LIN {X 0,Y 501.584,Z 1086.03,A -85,B 0,C 180,E1 12402.194,E2 12402.194} C_VEL
LIN {X 0,Y 502.565,Z 1075.07,A -85,B 0,C 180,E1 12406.965,E2 12406.965} C_VEL
LIN {X 0,Y 503.829,Z 1050.291,A -85,B 0,C 180,E1 12410.955,E2 12410.955} C_VEL
LIN {X 0,Y 505.175,Z 1014.827,A -85,B 0,C 180,E1 12413.746,E2 12413.746} C_VEL
LIN {X 0,Y 505.31,Z 972.689,A -85,B 0,C 180,E1 12415.098,E2 12415.098} C_VEL
LIN {X 0,Y 507.178,Z 860.099,A -85,B 0,C 180,E1 12417.103,E2 12417.103} C_VEL
LIN {X 0,Y 506.379,Z 795.398,A -85,B 0,C 180,E1 12419.992,E2 12419.992} C_VEL
LIN {X 0,Y 498.666,Z 762.06,A -85,B 0,C 180,E1 12422.013,E2 12422.013} C_VEL
LIN {X 0,Y 498.356,Z 762.06,A -85,B 0,C 180,E1 12431.466,E2 12431.466} C_VEL
LIN {X 0,Y 497.906,Z 762.06,A -85,B 0,C 180,E1 12441.773,E2 12441.773} C_VEL
LIN {X 0,Y 497.963,Z 763.805,A -85,B 0,C 180,E1 12445.471,E2 12445.471} C_VEL
LIN {X 0,Y 531.796,Z 813.89,A -85,B 0,C 180,E1 12453.677,E2 12453.677} C_VEL
LIN {X 0,Y 563.025,Z 870.759,A -85,B 0,C 180,E1 12459.883,E2 12459.883} C_VEL
LIN {X 0,Y 551.168,Z 956.836,A -85,B 0,C 180,E1 12463.133,E2 12463.133} C_VEL
LIN {X 0,Y 538.131,Z 1030.007,A -85,B 0,C 180,E1 12467.654,E2 12467.654} C_VEL
LIN {X 0,Y 525.784,Z 1080.484,A -85,B 0,C 180,E1 12472.6,E2 12472.6} C_VEL
LIN {X 0,Y 511.244,Z 1133.404,A -85,B 0,C 180,E1 12480.517,E2 12480.517} C_VEL
LIN {X 0,Y 502.991,Z 1174.818,A -85,B 0,C 180,E1 12489.75,E2 12489.75} C_VEL
LIN {X 0,Y 501.524,Z 1182.015,A -85,B 0,C 180,E1 12491.879,E2 12491.879} C_VEL
LIN {X 0,Y 492.392,Z 1193.006,A -85,B 0,C 180,E1 12495.627,E2 12495.627} C_VEL
LIN {X 0,Y 491.324,Z 1206.842,A -85,B 0,C 180,E1 12503.842,E2 12503.842} C_VEL
LIN {X 0,Y 491.082,Z 1209.864,A -85,B 0,C 180,E1 12510.932,E2 12510.932} C_VEL
LIN {X 0,Y 491.288,Z 1203.601,A -85,B 0,C 180,E1 12518.82,E2 12518.82} C_VEL
LIN {X 0,Y 493.711,Z 1183.881,A -85,B 0,C 180,E1 12527.78,E2 12527.78} C_VEL
LIN {X 0,Y 500.688,Z 1147.15,A -85,B 0,C 180,E1 12537.333,E2 12537.333} C_VEL
LIN {X 0,Y 514.987,Z 1096.477,A -85,B 0,C 180,E1 12546.035,E2 12546.035} C_VEL
LIN {X 0,Y 527.863,Z 1049.194,A -85,B 0,C 180,E1 12551.332,E2 12551.332} C_VEL
LIN {X 0,Y 540.974,Z 981.301,A -85,B 0,C 180,E1 12556.165,E2 12556.165} C_VEL
LIN {X 0,Y 554.262,Z 895.088,A -85,B 0,C 180,E1 12559.986,E2 12559.986} C_VEL
LIN {X 0,Y 555.637,Z 872.387,A -85,B 0,C 180,E1 12560.872,E2 12560.872} C_VEL
LIN {X 0,Y 528.213,Z 820.162,A -85,B 0,C 180,E1 12566.62,E2 12566.62} C_VEL
LIN {X 0,Y 497.316,Z 774.259,A -85,B 0,C 180,E1 12574.21,E2 12574.21} C_VEL
LIN {X 0,Y 489.979,Z 762.06,A -85,B 0,C 180,E1 12576.679,E2 12576.679} C_VEL
LIN {X 0,Y 490.167,Z 762.06,A -85,B 0,C 180,E1 12586.523,E2 12586.523} C_VEL
LIN {X 0,Y 490.448,Z 762.06,A -85,B 0,C 180,E1 12595.512,E2 12595.512} C_VEL
LIN {X 0,Y 490.543,Z 762.06,A -85,B 0,C 180,E1 12602.607,E2 12602.607} C_VEL
LIN {X 0,Y 490.241,Z 762.06,A -85,B 0,C 180,E1 12611.552,E2 12611.552} C_VEL
LIN {X 0,Y 489.948,Z 762.06,A -85,B 0,C 180,E1 12620.807,E2 12620.807} C_VEL
LIN {X 0,Y 490.069,Z 763.934,A -85,B 0,C 180,E1 12627.224,E2 12627.224} C_VEL
LIN {X 0,Y 516.661,Z 805.185,A -85,B 0,C 180,E1 12634.3,E2 12634.3} C_VEL
LIN {X 0,Y 534.44,Z 841.356,A -85,B 0,C 180,E1 12638.266,E2 12638.266} C_VEL
LIN {X 0,Y 545.43,Z 875.323,A -85,B 0,C 180,E1 12641.217,E2 12641.217} C_VEL
LIN {X 0,Y 533.055,Z 952.563,A -85,B 0,C 180,E1 12645.091,E2 12645.091} C_VEL
LIN {X 0,Y 517.932,Z 1030.736,A -85,B 0,C 180,E1 12651.287,E2 12651.287} C_VEL
LIN {X 0,Y 507.374,Z 1083.929,A -85,B 0,C 180,E1 12657.378,E2 12657.378} C_VEL
LIN {X 0,Y 498.428,Z 1126.212,A -85,B 0,C 180,E1 12664.723,E2 12664.723} C_VEL
LIN {X 0,Y 493.224,Z 1157.477,A -85,B 0,C 180,E1 12673.418,E2 12673.418} C_VEL
LIN {X 0,Y 491.274,Z 1174.671,A -85,B 0,C 180,E1 12681.963,E2 12681.963} C_VEL
LIN {X 0,Y 490.815,Z 1179.89,A -85,B 0,C 180,E1 12689.067,E2 12689.067} C_VEL
LIN {X 0,Y 491.301,Z 1175.791,A -85,B 0,C 180,E1 12697.049,E2 12697.049} C_VEL
LIN {X 0,Y 492.893,Z 1158.688,A -85,B 0,C 180,E1 12706.036,E2 12706.036} C_VEL
LIN {X 0,Y 497.85,Z 1128.291,A -85,B 0,C 180,E1 12714.725,E2 12714.725} C_VEL
LIN {X 0,Y 506.517,Z 1087.158,A -85,B 0,C 180,E1 12722.068,E2 12722.068} C_VEL
LIN {X 0,Y 517.427,Z 1033.436,A -85,B 0,C 180,E1 12728.362,E2 12728.362} C_VEL
LIN {X 0,Y 532.611,Z 955.706,A -85,B 0,C 180,E1 12734.592,E2 12734.592} C_VEL
LIN {X 0,Y 544.85,Z 880.188,A -85,B 0,C 180,E1 12738.499,E2 12738.499} C_VEL
LIN {X 0,Y 544.549,Z 868.405,A -85,B 0,C 180,E1 12739.16,E2 12739.16} C_VEL
LIN {X 0,Y 532.956,Z 841.944,A -85,B 0,C 180,E1 12741.803,E2 12741.803} C_VEL
LIN {X 0,Y 506.021,Z 868.419,A -85,B 0,C 180,E1 12744.215,E2 12744.215} C_VEL
LIN {X 0,Y 501.208,Z 875.563,A -85,B 0,C 180,E1 12744.507,E2 12744.507} C_VEL
LIN {X 0,Y 498.271,Z 876.326,A -85,B 0,C 180,E1 12745.014,E2 12745.014} C_VEL
LIN {X 0,Y 497.611,Z 997.367,A -85,B 0,C 180,E1 12747.209,E2 12747.209} C_VEL
LIN {X 0,Y 496.416,Z 1036.646,A -85,B 0,C 180,E1 12749.609,E2 12749.609} C_VEL
LIN {X 0,Y 494.731,Z 1066.862,A -85,B 0,C 180,E1 12753.356,E2 12753.356} C_VEL
LIN {X 0,Y 493.625,Z 1084.009,A -85,B 0,C 180,E1 12757.937,E2 12757.937} C_VEL
LIN {X 0,Y 493.732,Z 1086.304,A -85,B 0,C 180,E1 12763.08,E2 12763.08} C_VEL
LIN {X 0,Y 494.952,Z 1073.478,A -85,B 0,C 180,E1 12767.662,E2 12767.662} C_VEL
LIN {X 0,Y 496.219,Z 1046.852,A -85,B 0,C 180,E1 12771.59,E2 12771.59} C_VEL
LIN {X 0,Y 497.463,Z 1009.558,A -85,B 0,C 180,E1 12774.253,E2 12774.253} C_VEL
LIN {X 0,Y 497.511,Z 956.973,A -85,B 0,C 180,E1 12775.569,E2 12775.569} C_VEL
LIN {X 0,Y 499.597,Z 860.338,A -85,B 0,C 180,E1 12777.386,E2 12777.386} C_VEL
LIN {X 0,Y 498.988,Z 797.899,A -85,B 0,C 180,E1 12780.197,E2 12780.197} C_VEL
LIN {X 0,Y 490.711,Z 762.06,A -85,B 0,C 180,E1 12782.321,E2 12782.321} C_VEL
LIN {X 0,Y 490.334,Z 762.06,A -85,B 0,C 180,E1 12791.656,E2 12791.656} C_VEL
LIN {X 0,Y 489.914,Z 762.06,A -85,B 0,C 180,E1 12800.92,E2 12800.92} C_VEL
LIN {X 0,Y 489.97,Z 764.004,A -85,B 0,C 180,E1 12803.605,E2 12803.605} C_VEL
LIN {X 0,Y 519.882,Z 807.672,A -85,B 0,C 180,E1 12811.563,E2 12811.563} C_VEL
LIN {X 0,Y 553.961,Z 866.925,A -85,B 0,C 180,E1 12818.709,E2 12818.709} C_VEL
LIN {X 0,Y 556.724,Z 877.922,A -85,B 0,C 180,E1 12819.496,E2 12819.496} C_VEL
LIN {X 0,Y 544.196,Z 963.495,A -85,B 0,C 180,E1 12822.887,E2 12822.887} C_VEL
LIN {X 0,Y 530.49,Z 1037.128,A -85,B 0,C 180,E1 12827.636,E2 12827.636} C_VEL
LIN {X 0,Y 517.97,Z 1086.972,A -85,B 0,C 180,E1 12832.705,E2 12832.705} C_VEL
LIN {X 0,Y 502.88,Z 1138.745,A -85,B 0,C 180,E1 12840.976,E2 12840.976} C_VEL
LIN {X 0,Y 494.619,Z 1177.946,A -85,B 0,C 180,E1 12850.328,E2 12850.328} C_VEL
LIN {X 0,Y 492.392,Z 1193.006,A -85,B 0,C 180,E1 12855.627,E2 12855.627} C_VEL
LIN {X 0,Y 483.384,Z 1201.302,A -85,B 0,C 180,E1 12859.554,E2 12859.554} C_VEL
LIN {X 0,Y 483.111,Z 1209.384,A -85,B 0,C 180,E1 12867.348,E2 12867.348} C_VEL
LIN {X 0,Y 483.181,Z 1208.302,A -85,B 0,C 180,E1 12874.551,E2 12874.551} C_VEL
LIN {X 0,Y 483.898,Z 1196.27,A -85,B 0,C 180,E1 12883.159,E2 12883.159} C_VEL
LIN {X 0,Y 487.499,Z 1171.343,A -85,B 0,C 180,E1 12891.983,E2 12891.983} C_VEL
LIN {X 0,Y 498.347,Z 1129.563,A -85,B 0,C 180,E1 12901.42,E2 12901.42} C_VEL
LIN {X 0,Y 512.486,Z 1084.261,A -85,B 0,C 180,E1 12908.318,E2 12908.318} C_VEL
LIN {X 0,Y 526.188,Z 1028.475,A -85,B 0,C 180,E1 12913.62,E2 12913.62} C_VEL
LIN {X 0,Y 540.049,Z 953.551,A -85,B 0,C 180,E1 12918.185,E2 12918.185} C_VEL
LIN {X 0,Y 549.932,Z 876.36,A -85,B 0,C 180,E1 12921.343,E2 12921.343} C_VEL
LIN {X 0,Y 523.592,Z 825.389,A -85,B 0,C 180,E1 12927.097,E2 12927.097} C_VEL
LIN {X 0,Y 491.459,Z 776.33,A -85,B 0,C 180,E1 12935.431,E2 12935.431} C_VEL
LIN {X 0,Y 481.93,Z 762.06,A -85,B 0,C 180,E1 12938.717,E2 12938.717} C_VEL
LIN {X 0,Y 482.263,Z 762.06,A -85,B 0,C 180,E1 12948.146,E2 12948.146} C_VEL
LIN {X 0,Y 483.376,Z 762.06,A -85,B 0,C 180,E1 12959.048,E2 12959.048} C_VEL
LIN {X 0,Y 482.371,Z 762.06,A -85,B 0,C 180,E1 12969.908,E2 12969.908} C_VEL
LIN {X 0,Y 481.917,Z 762.06,A -85,B 0,C 180,E1 12979.248,E2 12979.248} C_VEL
LIN {X 0,Y 482.085,Z 763.893,A -85,B 0,C 180,E1 12985.251,E2 12985.251} C_VEL
LIN {X 0,Y 507.292,Z 802.31,A -85,B 0,C 180,E1 12992.639,E2 12992.639} C_VEL
LIN {X 0,Y 528.284,Z 842.326,A -85,B 0,C 180,E1 12997.503,E2 12997.503} C_VEL
LIN {X 0,Y 539.646,Z 877.144,A -85,B 0,C 180,E1 13000.663,E2 13000.663} C_VEL
LIN {X 0,Y 526.655,Z 954.407,A -85,B 0,C 180,E1 13004.611,E2 13004.611} C_VEL
LIN {X 0,Y 511.633,Z 1026.558,A -85,B 0,C 180,E1 13010.465,E2 13010.465} C_VEL
LIN {X 0,Y 499.546,Z 1085.365,A -85,B 0,C 180,E1 13017.24,E2 13017.24} C_VEL
LIN {X 0,Y 490.459,Z 1127.891,A -85,B 0,C 180,E1 13024.773,E2 13024.773} C_VEL
LIN {X 0,Y 485.168,Z 1158.664,A -85,B 0,C 180,E1 13033.602,E2 13033.602} C_VEL
LIN {X 0,Y 483.157,Z 1175.781,A -85,B 0,C 180,E1 13042.735,E2 13042.735} C_VEL
LIN {X 0,Y 483.141,Z 1179.887,A -85,B 0,C 180,E1 13050.852,E2 13050.852} C_VEL
LIN {X 0,Y 483.496,Z 1173.458,A -85,B 0,C 180,E1 13059.041,E2 13059.041} C_VEL
LIN {X 0,Y 485.186,Z 1154.94,A -85,B 0,C 180,E1 13067.662,E2 13067.662} C_VEL
LIN {X 0,Y 490.529,Z 1125.881,A -85,B 0,C 180,E1 13075.61,E2 13075.61} C_VEL
LIN {X 0,Y 499.831,Z 1082.617,A -85,B 0,C 180,E1 13083.082,E2 13083.082} C_VEL
LIN {X 0,Y 513.288,Z 1018.663,A -85,B 0,C 180,E1 13090.211,E2 13090.211} C_VEL
LIN {X 0,Y 527.819,Z 949.258,A -85,B 0,C 180,E1 13095.598,E2 13095.598} C_VEL
LIN {X 0,Y 539.307,Z 873.653,A -85,B 0,C 180,E1 13099.476,E2 13099.476} C_VEL
LIN {X 0,Y 529.886,Z 852.055,A -85,B 0,C 180,E1 13101.738,E2 13101.738} C_VEL
LIN {X 0,Y 506.285,Z 877.046,A -85,B 0,C 180,E1 13103.639,E2 13103.639} C_VEL
LIN {X 0,Y 497.175,Z 888.251,A -85,B 0,C 180,E1 13104.285,E2 13104.285} C_VEL
LIN {X 0,Y 492.723,Z 893.46,A -85,B 0,C 180,E1 13104.612,E2 13104.612} C_VEL
LIN {X 0,Y 490.436,Z 893.427,A -85,B 0,C 180,E1 13105.053,E2 13105.053} C_VEL
LIN {X 0,Y 489.824,Z 998.567,A -85,B 0,C 180,E1 13107.027,E2 13107.027} C_VEL
LIN {X 0,Y 488.596,Z 1038.169,A -85,B 0,C 180,E1 13109.498,E2 13109.498} C_VEL
LIN {X 0,Y 486.867,Z 1067.564,A -85,B 0,C 180,E1 13113.195,E2 13113.195} C_VEL
LIN {X 0,Y 485.76,Z 1084.332,A -85,B 0,C 180,E1 13117.561,E2 13117.561} C_VEL
LIN {X 0,Y 485.758,Z 1088.321,A -85,B 0,C 180,E1 13122.154,E2 13122.154} C_VEL
LIN {X 0,Y 486.785,Z 1077.934,A -85,B 0,C 180,E1 13126.994,E2 13126.994} C_VEL
LIN {X 0,Y 488.158,Z 1053.73,A -85,B 0,C 180,E1 13131.113,E2 13131.113} C_VEL
LIN {X 0,Y 489.686,Z 1018.309,A -85,B 0,C 180,E1 13134.05,E2 13134.05} C_VEL
LIN {X 0,Y 489.837,Z 975.895,A -85,B 0,C 180,E1 13135.5,E2 13135.5} C_VEL
LIN {X 0,Y 491.945,Z 862.053,A -85,B 0,C 180,E1 13137.621,E2 13137.621} C_VEL
LIN {X 0,Y 491.271,Z 799.056,A -85,B 0,C 180,E1 13140.485,E2 13140.485} C_VEL
LIN {X 0,Y 482.773,Z 762.06,A -85,B 0,C 180,E1 13142.755,E2 13142.755} C_VEL
LIN {X 0,Y 482.347,Z 762.06,A -85,B 0,C 180,E1 13151.852,E2 13151.852} C_VEL
LIN {X 0,Y 482.079,Z 764.083,A -85,B 0,C 180,E1 13161.564,E2 13161.564} C_VEL
LIN {X 0,Y 509.701,Z 804.062,A -85,B 0,C 180,E1 13169.658,E2 13169.658} C_VEL
LIN {X 0,Y 541.657,Z 858.159,A -85,B 0,C 180,E1 13176.848,E2 13176.848} C_VEL
LIN {X 0,Y 551.008,Z 880.185,A -85,B 0,C 180,E1 13178.953,E2 13178.953} C_VEL
LIN {X 0,Y 538.11,Z 964.302,A -85,B 0,C 180,E1 13182.341,E2 13182.341} C_VEL
LIN {X 0,Y 523.928,Z 1038.662,A -85,B 0,C 180,E1 13187.171,E2 13187.171} C_VEL
LIN {X 0,Y 510.351,Z 1092.222,A -85,B 0,C 180,E1 13192.688,E2 13192.688} C_VEL
LIN {X 0,Y 495.736,Z 1139.267,A -85,B 0,C 180,E1 13200.463,E2 13200.463} C_VEL
LIN {X 0,Y 486.53,Z 1179.412,A -85,B 0,C 180,E1 13210.462,E2 13210.462} C_VEL
LIN {X 0,Y 483.384,Z 1201.302,A -85,B 0,C 180,E1 13219.554,E2 13219.554} C_VEL
LIN {X 0,Y 475.339,Z 1206.85,A -85,B 0,C 180,E1 13223.646,E2 13223.646} C_VEL
LIN {X 0,Y 475.092,Z 1209.864,A -85,B 0,C 180,E1 13230.964,E2 13230.964} C_VEL
LIN {X 0,Y 475.378,Z 1203.447,A -85,B 0,C 180,E1 13239.232,E2 13239.232} C_VEL
LIN {X 0,Y 478.01,Z 1183.458,A -85,B 0,C 180,E1 13248.558,E2 13248.558} C_VEL
LIN {X 0,Y 486.538,Z 1146.276,A -85,B 0,C 180,E1 13258.706,E2 13258.706} C_VEL
LIN {X 0,Y 500.843,Z 1102.147,A -85,B 0,C 180,E1 13266.625,E2 13266.625} C_VEL
LIN {X 0,Y 515.281,Z 1049.016,A -85,B 0,C 180,E1 13272.527,E2 13272.527} C_VEL
LIN {X 0,Y 529.378,Z 979.214,A -85,B 0,C 180,E1 13277.472,E2 13277.472} C_VEL
LIN {X 0,Y 543.809,Z 890.869,A -85,B 0,C 180,E1 13281.365,E2 13281.365} C_VEL
LIN {X 0,Y 543.58,Z 878.558,A -85,B 0,C 180,E1 13281.993,E2 13281.993} C_VEL
LIN {X 0,Y 517.866,Z 828.802,A -85,B 0,C 180,E1 13287.841,E2 13287.841} C_VEL
LIN {X 0,Y 488.085,Z 783.083,A -85,B 0,C 180,E1 13295.863,E2 13295.863} C_VEL
LIN {X 0,Y 474.006,Z 762.06,A -85,B 0,C 180,E1 13301.263,E2 13301.263} C_VEL
LIN {X 0,Y 474.607,Z 762.06,A -85,B 0,C 180,E1 13311.675,E2 13311.675} C_VEL
LIN {X 0,Y 474.788,Z 762.06,A -85,B 0,C 180,E1 13320.862,E2 13320.862} C_VEL
LIN {X 0,Y 474.336,Z 762.06,A -85,B 0,C 180,E1 13330.078,E2 13330.078} C_VEL
LIN {X 0,Y 473.886,Z 762.06,A -85,B 0,C 180,E1 13339.587,E2 13339.587} C_VEL
LIN {X 0,Y 474.239,Z 764.161,A -85,B 0,C 180,E1 13343.078,E2 13343.078} C_VEL
LIN {X 0,Y 496.893,Z 797.841,A -85,B 0,C 180,E1 13350.511,E2 13350.511} C_VEL
LIN {X 0,Y 521.962,Z 842.457,A -85,B 0,C 180,E1 13356.636,E2 13356.636} C_VEL
LIN {X 0,Y 533.487,Z 882.016,A -85,B 0,C 180,E1 13360.213,E2 13360.213} C_VEL
LIN {X 0,Y 520.1,Z 957.236,A -85,B 0,C 180,E1 13364.177,E2 13364.177} C_VEL
LIN {X 0,Y 504.516,Z 1028.314,A -85,B 0,C 180,E1 13370.104,E2 13370.104} C_VEL
LIN {X 0,Y 490.514,Z 1092.461,A -85,B 0,C 180,E1 13377.966,E2 13377.966} C_VEL
LIN {X 0,Y 481.795,Z 1133.783,A -85,B 0,C 180,E1 13385.831,E2 13385.831} C_VEL
LIN {X 0,Y 476.551,Z 1162.076,A -85,B 0,C 180,E1 13394.721,E2 13394.721} C_VEL
LIN {X 0,Y 475.121,Z 1176.829,A -85,B 0,C 180,E1 13403.533,E2 13403.533} C_VEL
LIN {X 0,Y 475.143,Z 1179.884,A -85,B 0,C 180,E1 13410.866,E2 13410.866} C_VEL
LIN {X 0,Y 475.482,Z 1173.46,A -85,B 0,C 180,E1 13419.195,E2 13419.195} C_VEL
LIN {X 0,Y 477.332,Z 1154.919,A -85,B 0,C 180,E1 13427.962,E2 13427.962} C_VEL
LIN {X 0,Y 482.786,Z 1126.013,A -85,B 0,C 180,E1 13435.891,E2 13435.891} C_VEL
LIN {X 0,Y 491.966,Z 1083.974,A -85,B 0,C 180,E1 13443.208,E2 13443.208} C_VEL
LIN {X 0,Y 507.71,Z 1014.23,A -85,B 0,C 180,E1 13451.19,E2 13451.19} C_VEL
LIN {X 0,Y 523.097,Z 943.562,A -85,B 0,C 180,E1 13456.57,E2 13456.57} C_VEL
LIN {X 0,Y 533.311,Z 877.091,A -85,B 0,C 180,E1 13459.996,E2 13459.996} C_VEL
LIN {X 0,Y 528.067,Z 863.615,A -85,B 0,C 180,E1 13461.385,E2 13461.385} C_VEL
LIN {X 0,Y 510.923,Z 878.726,A -85,B 0,C 180,E1 13462.864,E2 13462.864} C_VEL
LIN {X 0,Y 484.538,Z 909.606,A -85,B 0,C 180,E1 13464.663,E2 13464.663} C_VEL
LIN {X 0,Y 482.579,Z 910.345,A -85,B 0,C 180,E1 13465.086,E2 13465.086} C_VEL
LIN {X 0,Y 481.993,Z 1000.898,A -85,B 0,C 180,E1 13466.888,E2 13466.888} C_VEL
LIN {X 0,Y 480.759,Z 1040.245,A -85,B 0,C 180,E1 13469.439,E2 13469.439} C_VEL
LIN {X 0,Y 478.974,Z 1069.26,A -85,B 0,C 180,E1 13473.203,E2 13473.203} C_VEL
LIN {X 0,Y 477.843,Z 1085.779,A -85,B 0,C 180,E1 13477.686,E2 13477.686} C_VEL
LIN {X 0,Y 477.87,Z 1089.18,A -85,B 0,C 180,E1 13482.501,E2 13482.501} C_VEL
LIN {X 0,Y 479.093,Z 1077.535,A -85,B 0,C 180,E1 13487.479,E2 13487.479} C_VEL
LIN {X 0,Y 480.432,Z 1053.615,A -85,B 0,C 180,E1 13491.426,E2 13491.426} C_VEL
LIN {X 0,Y 481.967,Z 1016.81,A -85,B 0,C 180,E1 13494.407,E2 13494.407} C_VEL
LIN {X 0,Y 482.09,Z 971.149,A -85,B 0,C 180,E1 13495.823,E2 13495.823} C_VEL
LIN {X 0,Y 484.377,Z 862.498,A -85,B 0,C 180,E1 13497.921,E2 13497.921} C_VEL
LIN {X 0,Y 483.697,Z 800.495,A -85,B 0,C 180,E1 13500.769,E2 13500.769} C_VEL
LIN {X 0,Y 474.792,Z 762.06,A -85,B 0,C 180,E1 13503.03,E2 13503.03} C_VEL
LIN {X 0,Y 474.221,Z 762.06,A -85,B 0,C 180,E1 13513.94,E2 13513.94} C_VEL
LIN {X 0,Y 474.16,Z 764.052,A -85,B 0,C 180,E1 13519.268,E2 13519.268} C_VEL
LIN {X 0,Y 499.405,Z 800.487,A -85,B 0,C 180,E1 13527.536,E2 13527.536} C_VEL
LIN {X 0,Y 530.576,Z 851.548,A -85,B 0,C 180,E1 13535.094,E2 13535.094} C_VEL
LIN {X 0,Y 545.17,Z 883.431,A -85,B 0,C 180,E1 13538.433,E2 13538.433} C_VEL
LIN {X 0,Y 531.635,Z 967.954,A -85,B 0,C 180,E1 13541.934,E2 13541.934} C_VEL
LIN {X 0,Y 517.137,Z 1040.86,A -85,B 0,C 180,E1 13546.77,E2 13546.77} C_VEL
LIN {X 0,Y 503.154,Z 1094.857,A -85,B 0,C 180,E1 13552.402,E2 13552.402} C_VEL
LIN {X 0,Y 489.557,Z 1136.821,A -85,B 0,C 180,E1 13559.298,E2 13559.298} C_VEL
LIN {X 0,Y 479.255,Z 1177.597,A -85,B 0,C 180,E1 13569.511,E2 13569.511} C_VEL
LIN {X 0,Y 475.526,Z 1200.714,A -85,B 0,C 180,E1 13579.012,E2 13579.012} C_VEL
LIN {X 0,Y 475.339,Z 1206.85,A -85,B 0,C 180,E1 13583.646,E2 13583.646} C_VEL
LIN {X 0,Y 467.171,Z 1209.532,A -85,B 0,C 180,E1 13587.823,E2 13587.823} C_VEL
LIN {X 0,Y 467.187,Z 1206.739,A -85,B 0,C 180,E1 13596.577,E2 13596.577} C_VEL
LIN {X 0,Y 468.325,Z 1193.121,A -85,B 0,C 180,E1 13605.073,E2 13605.073} C_VEL
LIN {X 0,Y 474.782,Z 1163.434,A -85,B 0,C 180,E1 13615.109,E2 13615.109} C_VEL
LIN {X 0,Y 488.029,Z 1122.377,A -85,B 0,C 180,E1 13624.124,E2 13624.124} C_VEL
LIN {X 0,Y 502.523,Z 1073.709,A -85,B 0,C 180,E1 13630.693,E2 13630.693} C_VEL
LIN {X 0,Y 516.474,Z 1015.511,A -85,B 0,C 180,E1 13635.758,E2 13635.758} C_VEL
LIN {X 0,Y 530.979,Z 939.661,A -85,B 0,C 180,E1 13640.052,E2 13640.052} C_VEL
LIN {X 0,Y 538.128,Z 882.914,A -85,B 0,C 180,E1 13642.435,E2 13642.435} C_VEL
LIN {X 0,Y 513.172,Z 833.711,A -85,B 0,C 180,E1 13648.356,E2 13648.356} C_VEL
LIN {X 0,Y 484.692,Z 789.71,A -85,B 0,C 180,E1 13656.297,E2 13656.297} C_VEL
LIN {X 0,Y 467.759,Z 767.034,A -85,B 0,C 180,E1 13662.666,E2 13662.666} C_VEL
LIN {X 0,Y 466.123,Z 762.06,A -85,B 0,C 180,E1 13663.978,E2 13663.978} C_VEL
LIN {X 0,Y 466.505,Z 762.06,A -85,B 0,C 180,E1 13673.409,E2 13673.409} C_VEL
LIN {X 0,Y 466.781,Z 762.06,A -85,B 0,C 180,E1 13680.877,E2 13680.877} C_VEL
LIN {X 0,Y 466.302,Z 762.06,A -85,B 0,C 180,E1 13690.254,E2 13690.254} C_VEL
LIN {X 0,Y 466.004,Z 763.552,A -85,B 0,C 180,E1 13700.367,E2 13700.367} C_VEL
LIN {X 0,Y 485.702,Z 792.496,A -85,B 0,C 180,E1 13707.882,E2 13707.882} C_VEL
LIN {X 0,Y 511.73,Z 836.107,A -85,B 0,C 180,E1 13714.862,E2 13714.862} C_VEL
LIN {X 0,Y 527.902,Z 883.432,A -85,B 0,C 180,E1 13719.615,E2 13719.615} C_VEL
LIN {X 0,Y 513.712,Z 959.705,A -85,B 0,C 180,E1 13723.704,E2 13723.704} C_VEL
LIN {X 0,Y 497.616,Z 1029.639,A -85,B 0,C 180,E1 13729.666,E2 13729.666} C_VEL
LIN {X 0,Y 482.651,Z 1093.729,A -85,B 0,C 180,E1 13737.84,E2 13737.84} C_VEL
LIN {X 0,Y 474.066,Z 1133.713,A -85,B 0,C 180,E1 13745.52,E2 13745.52} C_VEL
LIN {X 0,Y 468.702,Z 1162.094,A -85,B 0,C 180,E1 13754.458,E2 13754.458} C_VEL
LIN {X 0,Y 467.123,Z 1176.826,A -85,B 0,C 180,E1 13763.422,E2 13763.422} C_VEL
LIN {X 0,Y 467.143,Z 1179.88,A -85,B 0,C 180,E1 13770.881,E2 13770.881} C_VEL
LIN {X 0,Y 467.498,Z 1173.669,A -85,B 0,C 180,E1 13779.195,E2 13779.195} C_VEL
LIN {X 0,Y 469.312,Z 1156.084,A -85,B 0,C 180,E1 13787.836,E2 13787.836} C_VEL
LIN {X 0,Y 474.803,Z 1127.366,A -85,B 0,C 180,E1 13795.9,E2 13795.9} C_VEL
LIN {X 0,Y 483.948,Z 1086.113,A -85,B 0,C 180,E1 13803.22,E2 13803.22} C_VEL
LIN {X 0,Y 499.582,Z 1021.354,A -85,B 0,C 180,E1 13811.089,E2 13811.089} C_VEL
LIN {X 0,Y 515.411,Z 952.864,A -85,B 0,C 180,E1 13816.629,E2 13816.629} C_VEL
LIN {X 0,Y 527.262,Z 880.105,A -85,B 0,C 180,E1 13820.569,E2 13820.569} C_VEL
LIN {X 0,Y 523.154,Z 873.607,A -85,B 0,C 180,E1 13821.487,E2 13821.487} C_VEL
LIN {X 0,Y 477.184,Z 924.174,A -85,B 0,C 180,E1 13824.596,E2 13824.596} C_VEL
LIN {X 0,Y 474.757,Z 925.206,A -85,B 0,C 180,E1 13825.088,E2 13825.088} C_VEL
LIN {X 0,Y 474.205,Z 1002.132,A -85,B 0,C 180,E1 13826.703,E2 13826.703} C_VEL
LIN {X 0,Y 472.914,Z 1041.619,A -85,B 0,C 180,E1 13829.319,E2 13829.319} C_VEL
LIN {X 0,Y 471.025,Z 1071.154,A -85,B 0,C 180,E1 13833.255,E2 13833.255} C_VEL
LIN {X 0,Y 469.895,Z 1088.139,A -85,B 0,C 180,E1 13838.261,E2 13838.261} C_VEL
LIN {X 0,Y 470.017,Z 1089.721,A -85,B 0,C 180,E1 13843.167,E2 13843.167} C_VEL
LIN {X 0,Y 471.391,Z 1076.951,A -85,B 0,C 180,E1 13847.979,E2 13847.979} C_VEL
LIN {X 0,Y 472.845,Z 1050.905,A -85,B 0,C 180,E1 13852.026,E2 13852.026} C_VEL
LIN {X 0,Y 474.286,Z 1013.703,A -85,B 0,C 180,E1 13854.834,E2 13854.834} C_VEL
LIN {X 0,Y 474.389,Z 962.983,A -85,B 0,C 180,E1 13856.214,E2 13856.214} C_VEL
LIN {X 0,Y 476.785,Z 864.285,A -85,B 0,C 180,E1 13858.173,E2 13858.173} C_VEL
LIN {X 0,Y 476.244,Z 802.481,A -85,B 0,C 180,E1 13861.035,E2 13861.035} C_VEL
LIN {X 0,Y 466.791,Z 762.06,A -85,B 0,C 180,E1 13863.549,E2 13863.549} C_VEL
LIN {X 0,Y 466.169,Z 762.06,A -85,B 0,C 180,E1 13874.185,E2 13874.185} C_VEL
LIN {X 0,Y 466.279,Z 764.324,A -85,B 0,C 180,E1 13876.656,E2 13876.656} C_VEL
LIN {X 0,Y 486.502,Z 792.843,A -85,B 0,C 180,E1 13884.343,E2 13884.343} C_VEL
LIN {X 0,Y 515.657,Z 838.564,A -85,B 0,C 180,E1 13892.286,E2 13892.286} C_VEL
LIN {X 0,Y 539.433,Z 886.364,A -85,B 0,C 180,E1 13897.893,E2 13897.893} C_VEL
LIN {X 0,Y 525.485,Z 969.628,A -85,B 0,C 180,E1 13901.41,E2 13901.41} C_VEL
LIN {X 0,Y 510.287,Z 1043.422,A -85,B 0,C 180,E1 13906.39,E2 13906.39} C_VEL
LIN {X 0,Y 495.516,Z 1098.518,A -85,B 0,C 180,E1 13912.294,E2 13912.294} C_VEL
LIN {X 0,Y 481.866,Z 1140.041,A -85,B 0,C 180,E1 13919.259,E2 13919.259} C_VEL
LIN {X 0,Y 471.225,Z 1179.093,A -85,B 0,C 180,E1 13929.602,E2 13929.602} C_VEL
LIN {X 0,Y 467.574,Z 1200.713,A -85,B 0,C 180,E1 13938.823,E2 13938.823} C_VEL
LIN {X 0,Y 467.095,Z 1209.382,A -85,B 0,C 180,E1 13947.257,E2 13947.257} C_VEL
LIN {X 0,Y 467.171,Z 1209.532,A -85,B 0,C 180,E1 13947.823,E2 13947.823} C_VEL
LIN {X 0,Y 458.994,Z 1209.557,A -85,B 0,C 180,E1 13952.102,E2 13952.102} C_VEL
LIN {X 0,Y 459.664,Z 1201.987,A -85,B 0,C 180,E1 13960.511,E2 13960.511} C_VEL
LIN {X 0,Y 462.745,Z 1181.044,A -85,B 0,C 180,E1 13970.192,E2 13970.192} C_VEL
LIN {X 0,Y 473.775,Z 1143.968,A -85,B 0,C 180,E1 13980.615,E2 13980.615} C_VEL
LIN {X 0,Y 487.85,Z 1101.043,A -85,B 0,C 180,E1 13987.959,E2 13987.959} C_VEL
LIN {X 0,Y 503.176,Z 1046.685,A -85,B 0,C 180,E1 13993.929,E2 13993.929} C_VEL
LIN {X 0,Y 518.612,Z 974.719,A -85,B 0,C 180,E1 13998.951,E2 13998.951} C_VEL
LIN {X 0,Y 532.515,Z 886.798,A -85,B 0,C 180,E1 14002.934,E2 14002.934} C_VEL
LIN {X 0,Y 508.397,Z 838.738,A -85,B 0,C 180,E1 14008.892,E2 14008.892} C_VEL
LIN {X 0,Y 481.273,Z 796.244,A -85,B 0,C 180,E1 14016.734,E2 14016.734} C_VEL
LIN {X 0,Y 462.134,Z 769.028,A -85,B 0,C 180,E1 14024.554,E2 14024.554} C_VEL
LIN {X 0,Y 458.194,Z 762.06,A -85,B 0,C 180,E1 14027.513,E2 14027.513} C_VEL
LIN {X 0,Y 458.743,Z 762.06,A -85,B 0,C 180,E1 14037.101,E2 14037.101} C_VEL
LIN {X 0,Y 458.712,Z 762.06,A -85,B 0,C 180,E1 14046.592,E2 14046.592} C_VEL
LIN {X 0,Y 458.072,Z 763.44,A -85,B 0,C 180,E1 14057.223,E2 14057.223} C_VEL
LIN {X 0,Y 474.349,Z 787.339,A -85,B 0,C 180,E1 14064.765,E2 14064.765} C_VEL
LIN {X 0,Y 496.8,Z 822.569,A -85,B 0,C 180,E1 14071.742,E2 14071.742} C_VEL
LIN {X 0,Y 514.159,Z 858.855,A -85,B 0,C 180,E1 14076.35,E2 14076.35} C_VEL
LIN {X 0,Y 521.731,Z 889.332,A -85,B 0,C 180,E1 14079.19,E2 14079.19} C_VEL
LIN {X 0,Y 506.74,Z 964.951,A -85,B 0,C 180,E1 14083.414,E2 14083.414} C_VEL
LIN {X 0,Y 490.569,Z 1031.995,A -85,B 0,C 180,E1 14089.309,E2 14089.309} C_VEL
LIN {X 0,Y 475.745,Z 1090.626,A -85,B 0,C 180,E1 14097.015,E2 14097.015} C_VEL
LIN {X 0,Y 466.481,Z 1132.605,A -85,B 0,C 180,E1 14104.956,E2 14104.956} C_VEL
LIN {X 0,Y 461.112,Z 1160.952,A -85,B 0,C 180,E1 14113.706,E2 14113.706} C_VEL
LIN {X 0,Y 459.223,Z 1176.005,A -85,B 0,C 180,E1 14122.5,E2 14122.5} C_VEL
LIN {X 0,Y 459.172,Z 1179.877,A -85,B 0,C 180,E1 14130.896,E2 14130.896} C_VEL
LIN {X 0,Y 459.479,Z 1173.621,A -85,B 0,C 180,E1 14139.453,E2 14139.453} C_VEL
LIN {X 0,Y 461.466,Z 1155.987,A -85,B 0,C 180,E1 14148.149,E2 14148.149} C_VEL
LIN {X 0,Y 467.096,Z 1127.258,A -85,B 0,C 180,E1 14156.229,E2 14156.229} C_VEL
LIN {X 0,Y 477.468,Z 1082.296,A -85,B 0,C 180,E1 14164.208,E2 14164.208} C_VEL
LIN {X 0,Y 493.427,Z 1020.582,A -85,B 0,C 180,E1 14171.786,E2 14171.786} C_VEL
LIN {X 0,Y 509.695,Z 952.82,A -85,B 0,C 180,E1 14177.289,E2 14177.289} C_VEL
LIN {X 0,Y 522.118,Z 885.333,A -85,B 0,C 180,E1 14180.91,E2 14180.91} C_VEL
LIN {X 0,Y 517.116,Z 887.037,A -85,B 0,C 180,E1 14181.462,E2 14181.462} C_VEL
LIN {X 0,Y 476.926,Z 930.526,A -85,B 0,C 180,E1 14184.012,E2 14184.012} C_VEL
LIN {X 0,Y 469.128,Z 938.083,A -85,B 0,C 180,E1 14184.587,E2 14184.587} C_VEL
LIN {X 0,Y 466.787,Z 939.465,A -85,B 0,C 180,E1 14185.082,E2 14185.082} C_VEL
LIN {X 0,Y 466.381,Z 1005.04,A -85,B 0,C 180,E1 14186.592,E2 14186.592} C_VEL
LIN {X 0,Y 464.925,Z 1045.077,A -85,B 0,C 180,E1 14189.408,E2 14189.408} C_VEL
LIN {X 0,Y 463.087,Z 1074.12,A -85,B 0,C 180,E1 14193.555,E2 14193.555} C_VEL
LIN {X 0,Y 461.997,Z 1088.512,A -85,B 0,C 180,E1 14197.87,E2 14197.87} C_VEL
LIN {X 0,Y 462.085,Z 1091.124,A -85,B 0,C 180,E1 14202.9,E2 14202.9} C_VEL
LIN {X 0,Y 463.432,Z 1079.536,A -85,B 0,C 180,E1 14207.769,E2 14207.769} C_VEL
LIN {X 0,Y 465.008,Z 1053.975,A -85,B 0,C 180,E1 14212.002,E2 14212.002} C_VEL
LIN {X 0,Y 466.573,Z 1017.531,A -85,B 0,C 180,E1 14214.924,E2 14214.924} C_VEL
LIN {X 0,Y 466.676,Z 968.801,A -85,B 0,C 180,E1 14216.385,E2 14216.385} C_VEL
LIN {X 0,Y 469.254,Z 864.945,A -85,B 0,C 180,E1 14218.491,E2 14218.491} C_VEL
LIN {X 0,Y 468.788,Z 804.314,A -85,B 0,C 180,E1 14221.326,E2 14221.326} C_VEL
LIN {X 0,Y 458.821,Z 762.06,A -85,B 0,C 180,E1 14223.848,E2 14223.848} C_VEL
LIN {X 0,Y 458.434,Z 764.049,A -85,B 0,C 180,E1 14233.513,E2 14233.513} C_VEL
LIN {X 0,Y 474.874,Z 787.61,A -85,B 0,C 180,E1 14241.062,E2 14241.062} C_VEL
LIN {X 0,Y 499.584,Z 824.807,A -85,B 0,C 180,E1 14248.836,E2 14248.836} C_VEL
LIN {X 0,Y 528.571,Z 877.125,A -85,B 0,C 180,E1 14256.065,E2 14256.065} C_VEL
LIN {X 0,Y 533.404,Z 890.782,A -85,B 0,C 180,E1 14257.392,E2 14257.392} C_VEL
LIN {X 0,Y 519.07,Z 972.973,A -85,B 0,C 180,E1 14260.971,E2 14260.971} C_VEL
LIN {X 0,Y 503.555,Z 1045.32,A -85,B 0,C 180,E1 14265.953,E2 14265.953} C_VEL
LIN {X 0,Y 488.348,Z 1100.049,A -85,B 0,C 180,E1 14271.924,E2 14271.924} C_VEL
LIN {X 0,Y 474.11,Z 1143.306,A -85,B 0,C 180,E1 14279.255,E2 14279.255} C_VEL
LIN {X 0,Y 463.009,Z 1181.318,A -85,B 0,C 180,E1 14289.926,E2 14289.926} C_VEL
LIN {X 0,Y 459.407,Z 1202.144,A -85,B 0,C 180,E1 14299.585,E2 14299.585} C_VEL
LIN {X 0,Y 459.185,Z 1209.547,A -85,B 0,C 180,E1 14307.843,E2 14307.843} C_VEL
LIN {X 0,Y 458.994,Z 1209.557,A -85,B 0,C 180,E1 14312.102,E2 14312.102} C_VEL
LIN {X 0,Y 451.158,Z 1206.822,A -85,B 0,C 180,E1 14316.467,E2 14316.467} C_VEL
LIN {X 0,Y 452.584,Z 1193.142,A -85,B 0,C 180,E1 14325.611,E2 14325.611} C_VEL
LIN {X 0,Y 460.592,Z 1163.066,A -85,B 0,C 180,E1 14336.462,E2 14336.462} C_VEL
LIN {X 0,Y 473.251,Z 1125.481,A -85,B 0,C 180,E1 14344.751,E2 14344.751} C_VEL
LIN {X 0,Y 488.886,Z 1075.974,A -85,B 0,C 180,E1 14351.623,E2 14351.623} C_VEL
LIN {X 0,Y 504.174,Z 1016.605,A -85,B 0,C 180,E1 14356.938,E2 14356.938} C_VEL
LIN {X 0,Y 520.186,Z 937.476,A -85,B 0,C 180,E1 14361.431,E2 14361.431} C_VEL
LIN {X 0,Y 526.908,Z 890.491,A -85,B 0,C 180,E1 14363.445,E2 14363.445} C_VEL
LIN {X 0,Y 502.535,Z 841.787,A -85,B 0,C 180,E1 14369.719,E2 14369.719} C_VEL
LIN {X 0,Y 476.945,Z 801.367,A -85,B 0,C 180,E1 14377.5,E2 14377.5} C_VEL
LIN {X 0,Y 459.148,Z 776.049,A -85,B 0,C 180,E1 14385.104,E2 14385.104} C_VEL
LIN {X 0,Y 450.532,Z 762.06,A -85,B 0,C 180,E1 14391.226,E2 14391.226} C_VEL
LIN {X 0,Y 450.777,Z 762.06,A -85,B 0,C 180,E1 14400.908,E2 14400.908} C_VEL
LIN {X 0,Y 450.27,Z 762.06,A -85,B 0,C 180,E1 14410.623,E2 14410.623} C_VEL
LIN {X 0,Y 450.521,Z 764.588,A -85,B 0,C 180,E1 14413.515,E2 14413.515} C_VEL
LIN {X 0,Y 461.057,Z 779.073,A -85,B 0,C 180,E1 14419.961,E2 14419.961} C_VEL
LIN {X 0,Y 479.856,Z 807.091,A -85,B 0,C 180,E1 14427.42,E2 14427.42} C_VEL
LIN {X 0,Y 504.068,Z 849.498,A -85,B 0,C 180,E1 14434.297,E2 14434.297} C_VEL
LIN {X 0,Y 515.99,Z 892.827,A -85,B 0,C 180,E1 14438.657,E2 14438.657} C_VEL
LIN {X 0,Y 500.345,Z 967.933,A -85,B 0,C 180,E1 14442.953,E2 14442.953} C_VEL
LIN {X 0,Y 483.277,Z 1035.397,A -85,B 0,C 180,E1 14449.057,E2 14449.057} C_VEL
LIN {X 0,Y 468.003,Z 1092.824,A -85,B 0,C 180,E1 14456.89,E2 14456.89} C_VEL
LIN {X 0,Y 458.091,Z 1136.001,A -85,B 0,C 180,E1 14465.486,E2 14465.486} C_VEL
LIN {X 0,Y 452.527,Z 1164.387,A -85,B 0,C 180,E1 14474.885,E2 14474.885} C_VEL
LIN {X 0,Y 451.152,Z 1177.034,A -85,B 0,C 180,E1 14483.188,E2 14483.188} C_VEL
LIN {X 0,Y 451.175,Z 1180.109,A -85,B 0,C 180,E1 14490.912,E2 14490.912} C_VEL
LIN {X 0,Y 451.492,Z 1173.76,A -85,B 0,C 180,E1 14499.622,E2 14499.622} C_VEL
LIN {X 0,Y 453.644,Z 1155.821,A -85,B 0,C 180,E1 14508.473,E2 14508.473} C_VEL
LIN {X 0,Y 459.495,Z 1126.407,A -85,B 0,C 180,E1 14516.697,E2 14516.697} C_VEL
LIN {X 0,Y 472.089,Z 1075.964,A -85,B 0,C 180,E1 14525.683,E2 14525.683} C_VEL
LIN {X 0,Y 488.463,Z 1015.552,A -85,B 0,C 180,E1 14532.922,E2 14532.922} C_VEL
LIN {X 0,Y 505.573,Z 946.346,A -85,B 0,C 180,E1 14538.385,E2 14538.385} C_VEL
LIN {X 0,Y 513.431,Z 899.316,A -85,B 0,C 180,E1 14541.133,E2 14541.133} C_VEL
LIN {X 0,Y 469.372,Z 943.887,A -85,B 0,C 180,E1 14543.915,E2 14543.915} C_VEL
LIN {X 0,Y 459.702,Z 951.177,A -85,B 0,C 180,E1 14544.787,E2 14544.787} C_VEL
LIN {X 0,Y 458.4,Z 1013.796,A -85,B 0,C 180,E1 14546.764,E2 14546.764} C_VEL
LIN {X 0,Y 456.628,Z 1051.843,A -85,B 0,C 180,E1 14549.855,E2 14549.855} C_VEL
LIN {X 0,Y 454.952,Z 1078.875,A -85,B 0,C 180,E1 14554.262,E2 14554.262} C_VEL
LIN {X 0,Y 454.002,Z 1092.11,A -85,B 0,C 180,E1 14559.517,E2 14559.517} C_VEL
LIN {X 0,Y 454.413,Z 1090.629,A -85,B 0,C 180,E1 14564.264,E2 14564.264} C_VEL
LIN {X 0,Y 456.054,Z 1076.045,A -85,B 0,C 180,E1 14568.957,E2 14568.957} C_VEL
LIN {X 0,Y 457.647,Z 1047.994,A -85,B 0,C 180,E1 14572.961,E2 14572.961} C_VEL
LIN {X 0,Y 458.995,Z 1009.43,A -85,B 0,C 180,E1 14575.612,E2 14575.612} C_VEL
LIN {X 0,Y 460.471,Z 886.535,A -85,B 0,C 180,E1 14578.167,E2 14578.167} C_VEL
LIN {X 0,Y 462.946,Z 813.031,A -85,B 0,C 180,E1 14581.22,E2 14581.22} C_VEL
LIN {X 0,Y 450.833,Z 762.06,A -85,B 0,C 180,E1 14584.399,E2 14584.399} C_VEL
LIN {X 0,Y 450.505,Z 764.198,A -85,B 0,C 180,E1 14589.446,E2 14589.446} C_VEL
LIN {X 0,Y 461.273,Z 778.863,A -85,B 0,C 180,E1 14596.048,E2 14596.048} C_VEL
LIN {X 0,Y 483.678,Z 811.377,A -85,B 0,C 180,E1 14604.803,E2 14604.803} C_VEL
LIN {X 0,Y 512.958,Z 861.029,A -85,B 0,C 180,E1 14613.026,E2 14613.026} C_VEL
LIN {X 0,Y 527.764,Z 893.335,A -85,B 0,C 180,E1 14616.82,E2 14616.82} C_VEL
LIN {X 0,Y 512.702,Z 976.184,A -85,B 0,C 180,E1 14620.513,E2 14620.513} C_VEL
LIN {X 0,Y 497.038,Z 1046.381,A -85,B 0,C 180,E1 14625.435,E2 14625.435} C_VEL
LIN {X 0,Y 481.122,Z 1101.706,A -85,B 0,C 180,E1 14631.571,E2 14631.571} C_VEL
LIN {X 0,Y 466.239,Z 1145.92,A -85,B 0,C 180,E1 14639.222,E2 14639.222} C_VEL
LIN {X 0,Y 455.663,Z 1180.298,A -85,B 0,C 180,E1 14649.103,E2 14649.103} C_VEL
LIN {X 0,Y 451.44,Z 1202.009,A -85,B 0,C 180,E1 14659.399,E2 14659.399} C_VEL
LIN {X 0,Y 451.101,Z 1209.215,A -85,B 0,C 180,E1 14667.159,E2 14667.159} C_VEL
LIN {X 0,Y 451.169,Z 1208.12,A -85,B 0,C 180,E1 14674.874,E2 14674.874} C_VEL
LIN {X 0,Y 451.158,Z 1206.822,A -85,B 0,C 180,E1 14676.467,E2 14676.467} C_VEL
LIN {X 0,Y 443.709,Z 1201.77,A -85,B 0,C 180,E1 14680.874,E2 14680.874} C_VEL
LIN {X 0,Y 447.501,Z 1180.509,A -85,B 0,C 180,E1 14691.379,E2 14691.379} C_VEL
LIN {X 0,Y 457.612,Z 1149.611,A -85,B 0,C 180,E1 14700.517,E2 14700.517} C_VEL
LIN {X 0,Y 472.956,Z 1105.421,A -85,B 0,C 180,E1 14708.488,E2 14708.488} C_VEL
LIN {X 0,Y 489.835,Z 1050.109,A -85,B 0,C 180,E1 14714.859,E2 14714.859} C_VEL
LIN {X 0,Y 505.783,Z 981.05,A -85,B 0,C 180,E1 14719.886,E2 14719.886} C_VEL
LIN {X 0,Y 521.011,Z 893.036,A -85,B 0,C 180,E1 14724.072,E2 14724.072} C_VEL
LIN {X 0,Y 495.481,Z 842.575,A -85,B 0,C 180,E1 14730.944,E2 14730.944} C_VEL
LIN {X 0,Y 471.174,Z 804.242,A -85,B 0,C 180,E1 14738.826,E2 14738.826} C_VEL
LIN {X 0,Y 455.122,Z 781.727,A -85,B 0,C 180,E1 14746.202,E2 14746.202} C_VEL
LIN {X 0,Y 446.56,Z 769.011,A -85,B 0,C 180,E1 14752.622,E2 14752.622} C_VEL
LIN {X 0,Y 443.325,Z 762.06,A -85,B 0,C 180,E1 14758.962,E2 14758.962} C_VEL
LIN {X 0,Y 443.065,Z 764.606,A -85,B 0,C 180,E1 14767.135,E2 14767.135} C_VEL
LIN {X 0,Y 448.782,Z 773.124,A -85,B 0,C 180,E1 14773.693,E2 14773.693} C_VEL
LIN {X 0,Y 458.922,Z 787.235,A -85,B 0,C 180,E1 14779.927,E2 14779.927} C_VEL
LIN {X 0,Y 477.771,Z 815.557,A -85,B 0,C 180,E1 14787.471,E2 14787.471} C_VEL
LIN {X 0,Y 501.293,Z 858.84,A -85,B 0,C 180,E1 14794.383,E2 14794.383} C_VEL
LIN {X 0,Y 510.388,Z 895.709,A -85,B 0,C 180,E1 14798.086,E2 14798.086} C_VEL
LIN {X 0,Y 493.979,Z 970.968,A -85,B 0,C 180,E1 14802.482,E2 14802.482} C_VEL
LIN {X 0,Y 476.368,Z 1037.496,A -85,B 0,C 180,E1 14808.65,E2 14808.65} C_VEL
LIN {X 0,Y 460.702,Z 1093.448,A -85,B 0,C 180,E1 14816.459,E2 14816.459} C_VEL
LIN {X 0,Y 449.948,Z 1137.478,A -85,B 0,C 180,E1 14825.579,E2 14825.579} C_VEL
LIN {X 0,Y 444.672,Z 1164.354,A -85,B 0,C 180,E1 14834.612,E2 14834.612} C_VEL
LIN {X 0,Y 443.183,Z 1177.211,A -85,B 0,C 180,E1 14843.065,E2 14843.065} C_VEL
LIN {X 0,Y 443.177,Z 1180.319,A -85,B 0,C 180,E1 14850.929,E2 14850.929} C_VEL
LIN {X 0,Y 443.516,Z 1173.907,A -85,B 0,C 180,E1 14859.797,E2 14859.797} C_VEL
LIN {X 0,Y 445.805,Z 1155.657,A -85,B 0,C 180,E1 14868.81,E2 14868.81} C_VEL
LIN {X 0,Y 452.151,Z 1124.848,A -85,B 0,C 180,E1 14877.345,E2 14877.345} C_VEL
LIN {X 0,Y 465.104,Z 1076.489,A -85,B 0,C 180,E1 14886.188,E2 14886.188} C_VEL
LIN {X 0,Y 482.27,Z 1016.004,A -85,B 0,C 180,E1 14893.543,E2 14893.543} C_VEL
LIN {X 0,Y 499.801,Z 947.723,A -85,B 0,C 180,E1 14898.996,E2 14898.996} C_VEL
LIN {X 0,Y 506.516,Z 916.298,A -85,B 0,C 180,E1 14900.807,E2 14900.807} C_VEL
LIN {X 0,Y 454.799,Z 962.104,A -85,B 0,C 180,E1 14904.35,E2 14904.35} C_VEL
LIN {X 0,Y 451.126,Z 963.3,A -85,B 0,C 180,E1 14904.988,E2 14904.988} C_VEL
LIN {X 0,Y 450.644,Z 1013.525,A -85,B 0,C 180,E1 14906.488,E2 14906.488} C_VEL
LIN {X 0,Y 448.904,Z 1051.356,A -85,B 0,C 180,E1 14909.527,E2 14909.527} C_VEL
LIN {X 0,Y 447.157,Z 1078.893,A -85,B 0,C 180,E1 14913.938,E2 14913.938} C_VEL
LIN {X 0,Y 446.088,Z 1092.75,A -85,B 0,C 180,E1 14919.146,E2 14919.146} C_VEL
LIN {X 0,Y 446.503,Z 1091.849,A -85,B 0,C 180,E1 14924.286,E2 14924.286} C_VEL
LIN {X 0,Y 448.331,Z 1076.007,A -85,B 0,C 180,E1 14929.331,E2 14929.331} C_VEL
LIN {X 0,Y 449.969,Z 1048.084,A -85,B 0,C 180,E1 14933.279,E2 14933.279} C_VEL
LIN {X 0,Y 451.332,Z 1008.239,A -85,B 0,C 180,E1 14935.96,E2 14935.96} C_VEL
LIN {X 0,Y 454.277,Z 866.312,A -85,B 0,C 180,E1 14939.165,E2 14939.165} C_VEL
LIN {X 0,Y 453.886,Z 807.63,A -85,B 0,C 180,E1 14941.972,E2 14941.972} C_VEL
LIN {X 0,Y 443.955,Z 766.122,A -85,B 0,C 180,E1 14944.713,E2 14944.713} C_VEL
LIN {X 0,Y 449.283,Z 773.693,A -85,B 0,C 180,E1 14950.024,E2 14950.024} C_VEL
LIN {X 0,Y 458.857,Z 786.417,A -85,B 0,C 180,E1 14955.827,E2 14955.827} C_VEL
LIN {X 0,Y 480.721,Z 818.795,A -85,B 0,C 180,E1 14964.593,E2 14964.593} C_VEL
LIN {X 0,Y 508.896,Z 867.656,A -85,B 0,C 180,E1 14972.77,E2 14972.77} C_VEL
LIN {X 0,Y 521.883,Z 897.23,A -85,B 0,C 180,E1 14976.289,E2 14976.289} C_VEL
LIN {X 0,Y 506.537,Z 978.252,A -85,B 0,C 180,E1 14979.984,E2 14979.984} C_VEL
LIN {X 0,Y 490.621,Z 1047.207,A -85,B 0,C 180,E1 14984.882,E2 14984.882} C_VEL
LIN {X 0,Y 473.937,Z 1103.013,A -85,B 0,C 180,E1 14991.181,E2 14991.181} C_VEL
LIN {X 0,Y 458.667,Z 1147.074,A -85,B 0,C 180,E1 14998.934,E2 14998.934} C_VEL
LIN {X 0,Y 448.311,Z 1179.044,A -85,B 0,C 180,E1 15008.092,E2 15008.092} C_VEL
LIN {X 0,Y 443.789,Z 1200.471,A -85,B 0,C 180,E1 15018.215,E2 15018.215} C_VEL
LIN {X 0,Y 443.125,Z 1208.982,A -85,B 0,C 180,E1 15027.108,E2 15027.108} C_VEL
LIN {X 0,Y 443.141,Z 1206.717,A -85,B 0,C 180,E1 15036.475,E2 15036.475} C_VEL
LIN {X 0,Y 443.709,Z 1201.77,A -85,B 0,C 180,E1 15040.874,E2 15040.874} C_VEL
LIN {X 0,Y 436.472,Z 1194.949,A -85,B 0,C 180,E1 15045.318,E2 15045.318} C_VEL
LIN {X 0,Y 443.943,Z 1168.908,A -85,B 0,C 180,E1 15055.892,E2 15055.892} C_VEL
LIN {X 0,Y 457.507,Z 1130.431,A -85,B 0,C 180,E1 15064.958,E2 15064.958} C_VEL
LIN {X 0,Y 474.339,Z 1081.138,A -85,B 0,C 180,E1 15072.246,E2 15072.246} C_VEL
LIN {X 0,Y 491.27,Z 1021.137,A -85,B 0,C 180,E1 15077.897,E2 15077.897} C_VEL
LIN {X 0,Y 508.187,Z 943.293,A -85,B 0,C 180,E1 15082.498,E2 15082.498} C_VEL
LIN {X 0,Y 515.281,Z 896.132,A -85,B 0,C 180,E1 15084.664,E2 15084.664} C_VEL
LIN {X 0,Y 489.738,Z 845.891,A -85,B 0,C 180,E1 15091.81,E2 15091.81} C_VEL
LIN {X 0,Y 467.228,Z 809.997,A -85,B 0,C 180,E1 15099.51,E2 15099.51} C_VEL
LIN {X 0,Y 450.071,Z 784.337,A -85,B 0,C 180,E1 15108.273,E2 15108.273} C_VEL
LIN {X 0,Y 443.191,Z 775.76,A -85,B 0,C 180,E1 15114.047,E2 15114.047} C_VEL
LIN {X 0,Y 440.801,Z 769.64,A -85,B 0,C 180,E1 15118.956,E2 15118.956} C_VEL
LIN {X 0,Y 441.156,Z 772.486,A -85,B 0,C 180,E1 15127.104,E2 15127.104} C_VEL
LIN {X 0,Y 446.935,Z 781.296,A -85,B 0,C 180,E1 15133.813,E2 15133.813} C_VEL
LIN {X 0,Y 460.027,Z 799.205,A -85,B 0,C 180,E1 15141.403,E2 15141.403} C_VEL
LIN {X 0,Y 481.951,Z 834.89,A -85,B 0,C 180,E1 15149.535,E2 15149.535} C_VEL
LIN {X 0,Y 499.001,Z 871.192,A -85,B 0,C 180,E1 15154.753,E2 15154.753} C_VEL
LIN {X 0,Y 504.595,Z 899.61,A -85,B 0,C 180,E1 15157.551,E2 15157.551} C_VEL
LIN {X 0,Y 487.331,Z 975.426,A -85,B 0,C 180,E1 15162.106,E2 15162.106} C_VEL
LIN {X 0,Y 469.02,Z 1041.027,A -85,B 0,C 180,E1 15168.39,E2 15168.39} C_VEL
LIN {X 0,Y 452.919,Z 1096.308,A -85,B 0,C 180,E1 15176.382,E2 15176.382} C_VEL
LIN {X 0,Y 441.892,Z 1138.662,A -85,B 0,C 180,E1 15185.596,E2 15185.596} C_VEL
LIN {X 0,Y 436.549,Z 1165.383,A -85,B 0,C 180,E1 15194.835,E2 15194.835} C_VEL
LIN {X 0,Y 435.206,Z 1177.483,A -85,B 0,C 180,E1 15203.01,E2 15203.01} C_VEL
LIN {X 0,Y 435.18,Z 1180.566,A -85,B 0,C 180,E1 15210.946,E2 15210.946} C_VEL
LIN {X 0,Y 435.546,Z 1174.062,A -85,B 0,C 180,E1 15219.978,E2 15219.978} C_VEL
LIN {X 0,Y 437.778,Z 1156.529,A -85,B 0,C 180,E1 15228.747,E2 15228.747} C_VEL
LIN {X 0,Y 444.698,Z 1124.602,A -85,B 0,C 180,E1 15237.843,E2 15237.843} C_VEL
LIN {X 0,Y 458.358,Z 1076.479,A -85,B 0,C 180,E1 15246.807,E2 15246.807} C_VEL
LIN {X 0,Y 476.305,Z 1015.789,A -85,B 0,C 180,E1 15254.255,E2 15254.255} C_VEL
LIN {X 0,Y 494.539,Z 947.282,A -85,B 0,C 180,E1 15259.746,E2 15259.746} C_VEL
LIN {X 0,Y 498.508,Z 929.754,A -85,B 0,C 180,E1 15260.802,E2 15260.802} C_VEL
LIN {X 0,Y 455.096,Z 967.517,A -85,B 0,C 180,E1 15263.609,E2 15263.609} C_VEL
LIN {X 0,Y 443.943,Z 974.497,A -85,B 0,C 180,E1 15264.735,E2 15264.735} C_VEL
LIN {X 0,Y 442.444,Z 1025.954,A -85,B 0,C 180,E1 15266.984,E2 15266.984} C_VEL
LIN {X 0,Y 440.185,Z 1062.43,A -85,B 0,C 180,E1 15270.653,E2 15270.653} C_VEL
LIN {X 0,Y 438.634,Z 1086.042,A -85,B 0,C 180,E1 15275.483,E2 15275.483} C_VEL
LIN {X 0,Y 438.189,Z 1095.186,A -85,B 0,C 180,E1 15280.857,E2 15280.857} C_VEL
LIN {X 0,Y 439.079,Z 1089.427,A -85,B 0,C 180,E1 15286.128,E2 15286.128} C_VEL
LIN {X 0,Y 441.062,Z 1069.412,A -85,B 0,C 180,E1 15290.904,E2 15290.904} C_VEL
LIN {X 0,Y 442.87,Z 1036.614,A -85,B 0,C 180,E1 15294.611,E2 15294.611} C_VEL
LIN {X 0,Y 443.746,Z 993.821,A -85,B 0,C 180,E1 15296.75,E2 15296.75} C_VEL
LIN {X 0,Y 446.71,Z 868.251,A -85,B 0,C 180,E1 15299.468,E2 15299.468} C_VEL
LIN {X 0,Y 446.534,Z 809.66,A -85,B 0,C 180,E1 15302.296,E2 15302.296} C_VEL
LIN {X 0,Y 440.557,Z 779.177,A -85,B 0,C 180,E1 15304.43,E2 15304.43} C_VEL
LIN {X 0,Y 442.015,Z 775.369,A -85,B 0,C 180,E1 15304.981,E2 15304.981} C_VEL
LIN {X 0,Y 446.775,Z 780.607,A -85,B 0,C 180,E1 15309.526,E2 15309.526} C_VEL
LIN {X 0,Y 456.585,Z 794.353,A -85,B 0,C 180,E1 15315.722,E2 15315.722} C_VEL
LIN {X 0,Y 477.487,Z 825.821,A -85,B 0,C 180,E1 15324.317,E2 15324.317} C_VEL
LIN {X 0,Y 504.727,Z 874.104,A -85,B 0,C 180,E1 15332.499,E2 15332.499} C_VEL
LIN {X 0,Y 515.991,Z 901.364,A -85,B 0,C 180,E1 15335.751,E2 15335.751} C_VEL
LIN {X 0,Y 499.974,Z 982.588,A -85,B 0,C 180,E1 15339.572,E2 15339.572} C_VEL
LIN {X 0,Y 483.809,Z 1049.534,A -85,B 0,C 180,E1 15344.459,E2 15344.459} C_VEL
LIN {X 0,Y 466.853,Z 1103.957,A -85,B 0,C 180,E1 15350.735,E2 15350.735} C_VEL
LIN {X 0,Y 451.094,Z 1148.073,A -85,B 0,C 180,E1 15358.636,E2 15358.636} C_VEL
LIN {X 0,Y 440.551,Z 1179.709,A -85,B 0,C 180,E1 15367.794,E2 15367.794} C_VEL
LIN {X 0,Y 435.548,Z 1201.786,A -85,B 0,C 180,E1 15379.007,E2 15379.007} C_VEL
LIN {X 0,Y 435.12,Z 1208.721,A -85,B 0,C 180,E1 15387.055,E2 15387.055} C_VEL
LIN {X 0,Y 435.138,Z 1207.114,A -85,B 0,C 180,E1 15395.863,E2 15395.863} C_VEL
LIN {X 0,Y 436.472,Z 1194.949,A -85,B 0,C 180,E1 15405.318,E2 15405.318} C_VEL
LIN {X 0,Y 430.823,Z 1186.666,A -85,B 0,C 180,E1 15409.837,E2 15409.837} C_VEL
LIN {X 0,Y 440.133,Z 1157.837,A -85,B 0,C 180,E1 15419.484,E2 15419.484} C_VEL
LIN {X 0,Y 455.851,Z 1115.725,A -85,B 0,C 180,E1 15428.073,E2 15428.073} C_VEL
LIN {X 0,Y 473.937,Z 1062.087,A -85,B 0,C 180,E1 15434.965,E2 15434.965} C_VEL
LIN {X 0,Y 490.309,Z 1000.156,A -85,B 0,C 180,E1 15440.04,E2 15440.04} C_VEL
LIN {X 0,Y 508.698,Z 912.565,A -85,B 0,C 180,E1 15444.534,E2 15444.534} C_VEL
LIN {X 0,Y 509.759,Z 900.065,A -85,B 0,C 180,E1 15445.185,E2 15445.185} C_VEL
LIN {X 0,Y 484.307,Z 849.219,A -85,B 0,C 180,E1 15452.671,E2 15452.671} C_VEL
LIN {X 0,Y 461.504,Z 812.447,A -85,B 0,C 180,E1 15461.005,E2 15461.005} C_VEL
LIN {X 0,Y 446.663,Z 790.942,A -85,B 0,C 180,E1 15469.174,E2 15469.174} C_VEL
LIN {X 0,Y 441.332,Z 783.565,A -85,B 0,C 180,E1 15474.022,E2 15474.022} C_VEL
LIN {X 0,Y 438.386,Z 777.393,A -85,B 0,C 180,E1 15480.933,E2 15480.933} C_VEL
LIN {X 0,Y 439.412,Z 780.827,A -85,B 0,C 180,E1 15487.506,E2 15487.506} C_VEL
LIN {X 0,Y 445.04,Z 789.346,A -85,B 0,C 180,E1 15493.873,E2 15493.873} C_VEL
LIN {X 0,Y 458.271,Z 808.441,A -85,B 0,C 180,E1 15501.616,E2 15501.616} C_VEL
LIN {X 0,Y 478.813,Z 842.196,A -85,B 0,C 180,E1 15509.303,E2 15509.303} C_VEL
LIN {X 0,Y 494.398,Z 877.15,A -85,B 0,C 180,E1 15514.397,E2 15514.397} C_VEL
LIN {X 0,Y 498.879,Z 903.323,A -85,B 0,C 180,E1 15516.992,E2 15516.992} C_VEL
LIN {X 0,Y 481.354,Z 977.266,A -85,B 0,C 180,E1 15521.519,E2 15521.519} C_VEL
LIN {X 0,Y 462.173,Z 1043.114,A -85,B 0,C 180,E1 15527.949,E2 15527.949} C_VEL
LIN {X 0,Y 445.501,Z 1097.894,A -85,B 0,C 180,E1 15536.068,E2 15536.068} C_VEL
LIN {X 0,Y 433.922,Z 1139.986,A -85,B 0,C 180,E1 15545.559,E2 15545.559} C_VEL
LIN {X 0,Y 428.443,Z 1166.351,A -85,B 0,C 180,E1 15555.066,E2 15555.066} C_VEL
LIN {X 0,Y 427.222,Z 1177.623,A -85,B 0,C 180,E1 15562.805,E2 15562.805} C_VEL
LIN {X 0,Y 427.211,Z 1180.828,A -85,B 0,C 180,E1 15570.964,E2 15570.964} C_VEL
LIN {X 0,Y 427.558,Z 1174.212,A -85,B 0,C 180,E1 15580.166,E2 15580.166} C_VEL
LIN {X 0,Y 429.994,Z 1156.214,A -85,B 0,C 180,E1 15589.135,E2 15589.135} C_VEL
LIN {X 0,Y 437.83,Z 1123.134,A -85,B 0,C 180,E1 15598.681,E2 15598.681} C_VEL
LIN {X 0,Y 452.228,Z 1074.859,A -85,B 0,C 180,E1 15607.694,E2 15607.694} C_VEL
LIN {X 0,Y 471.366,Z 1012.664,A -85,B 0,C 180,E1 15615.276,E2 15615.276} C_VEL
LIN {X 0,Y 489.962,Z 944.278,A -85,B 0,C 180,E1 15620.661,E2 15620.661} C_VEL
LIN {X 0,Y 444.257,Z 980.339,A -85,B 0,C 180,E1 15623.835,E2 15623.835} C_VEL
LIN {X 0,Y 435.93,Z 984.623,A -85,B 0,C 180,E1 15624.789,E2 15624.789} C_VEL
LIN {X 0,Y 434.445,Z 1032.398,A -85,B 0,C 180,E1 15627.2,E2 15627.2} C_VEL
LIN {X 0,Y 432.138,Z 1067.372,A -85,B 0,C 180,E1 15631.115,E2 15631.115} C_VEL
LIN {X 0,Y 430.549,Z 1089.219,A -85,B 0,C 180,E1 15636.157,E2 15636.157} C_VEL
LIN {X 0,Y 430.298,Z 1096.297,A -85,B 0,C 180,E1 15641.682,E2 15641.682} C_VEL
LIN {X 0,Y 431.436,Z 1089.03,A -85,B 0,C 180,E1 15646.847,E2 15646.847} C_VEL
LIN {X 0,Y 433.467,Z 1068.107,A -85,B 0,C 180,E1 15651.504,E2 15651.504} C_VEL
LIN {X 0,Y 435.459,Z 1033.634,A -85,B 0,C 180,E1 15655.187,E2 15655.187} C_VEL
LIN {X 0,Y 436.123,Z 991.941,A -85,B 0,C 180,E1 15657.13,E2 15657.13} C_VEL
LIN {X 0,Y 439.244,Z 869.764,A -85,B 0,C 180,E1 15659.813,E2 15659.813} C_VEL
LIN {X 0,Y 439.137,Z 811.292,A -85,B 0,C 180,E1 15662.668,E2 15662.668} C_VEL
LIN {X 0,Y 436.47,Z 794.192,A -85,B 0,C 180,E1 15663.997,E2 15663.997} C_VEL
LIN {X 0,Y 440.646,Z 783.184,A -85,B 0,C 180,E1 15665.492,E2 15665.492} C_VEL
LIN {X 0,Y 445.941,Z 790.196,A -85,B 0,C 180,E1 15670.41,E2 15670.41} C_VEL
LIN {X 0,Y 458.859,Z 808.832,A -85,B 0,C 180,E1 15677.868,E2 15677.868} C_VEL
LIN {X 0,Y 481.451,Z 844.996,A -85,B 0,C 180,E1 15686.488,E2 15686.488} C_VEL
LIN {X 0,Y 506.635,Z 893.495,A -85,B 0,C 180,E1 15693.963,E2 15693.963} C_VEL
LIN {X 0,Y 510.18,Z 905.245,A -85,B 0,C 180,E1 15695.205,E2 15695.205} C_VEL
LIN {X 0,Y 493.435,Z 986.925,A -85,B 0,C 180,E1 15699.142,E2 15699.142} C_VEL
LIN {X 0,Y 476.811,Z 1052.514,A -85,B 0,C 180,E1 15704.089,E2 15704.089} C_VEL
LIN {X 0,Y 459.056,Z 1107.082,A -85,B 0,C 180,E1 15710.596,E2 15710.596} C_VEL
LIN {X 0,Y 442.626,Z 1151.59,A -85,B 0,C 180,E1 15718.97,E2 15718.97} C_VEL
LIN {X 0,Y 431.699,Z 1184.273,A -85,B 0,C 180,E1 15729.146,E2 15729.146} C_VEL
LIN {X 0,Y 427.412,Z 1202.97,A -85,B 0,C 180,E1 15739.831,E2 15739.831} C_VEL
LIN {X 0,Y 427.512,Z 1208.952,A -85,B 0,C 180,E1 15749.037,E2 15749.037} C_VEL
LIN {X 0,Y 427.199,Z 1205.986,A -85,B 0,C 180,E1 15757.196,E2 15757.196} C_VEL
LIN {X 0,Y 429.642,Z 1191.481,A -85,B 0,C 180,E1 15767.525,E2 15767.525} C_VEL
LIN {X 0,Y 430.823,Z 1186.666,A -85,B 0,C 180,E1 15769.837,E2 15769.837} C_VEL
LIN {X 0,Y 425.975,Z 1176.329,A -85,B 0,C 180,E1 15774.335,E2 15774.335} C_VEL
LIN {X 0,Y 439.185,Z 1140.817,A -85,B 0,C 180,E1 15783.992,E2 15783.992} C_VEL
LIN {X 0,Y 457.186,Z 1093.239,A -85,B 0,C 180,E1 15791.971,E2 15791.971} C_VEL
LIN {X 0,Y 475.654,Z 1035.566,A -85,B 0,C 180,E1 15798.098,E2 15798.098} C_VEL
LIN {X 0,Y 493.595,Z 961.845,A -85,B 0,C 180,E1 15802.971,E2 15802.971} C_VEL
LIN {X 0,Y 504.601,Z 904.966,A -85,B 0,C 180,E1 15805.608,E2 15805.608} C_VEL
LIN {X 0,Y 479.969,Z 854.746,A -85,B 0,C 180,E1 15813.167,E2 15813.167} C_VEL
LIN {X 0,Y 458.248,Z 819.09,A -85,B 0,C 180,E1 15821.46,E2 15821.46} C_VEL
LIN {X 0,Y 444.147,Z 798.183,A -85,B 0,C 180,E1 15829.548,E2 15829.548} C_VEL
LIN {X 0,Y 438.854,Z 790.845,A -85,B 0,C 180,E1 15834.61,E2 15834.61} C_VEL
LIN {X 0,Y 436.45,Z 785.129,A -85,B 0,C 180,E1 15840.938,E2 15840.938} C_VEL
LIN {X 0,Y 437.471,Z 788.671,A -85,B 0,C 180,E1 15847.539,E2 15847.539} C_VEL
LIN {X 0,Y 443.233,Z 797.551,A -85,B 0,C 180,E1 15854.057,E2 15854.057} C_VEL
LIN {X 0,Y 456.779,Z 817.679,A -85,B 0,C 180,E1 15861.946,E2 15861.946} C_VEL
LIN {X 0,Y 477.36,Z 852.651,A -85,B 0,C 180,E1 15869.65,E2 15869.65} C_VEL
LIN {X 0,Y 490.292,Z 885.449,A -85,B 0,C 180,E1 15874.277,E2 15874.277} C_VEL
LIN {X 0,Y 493.097,Z 907.755,A -85,B 0,C 180,E1 15876.462,E2 15876.462} C_VEL
LIN {X 0,Y 474.845,Z 981.298,A -85,B 0,C 180,E1 15881.084,E2 15881.084} C_VEL
LIN {X 0,Y 454.703,Z 1047.26,A -85,B 0,C 180,E1 15887.743,E2 15887.743} C_VEL
LIN {X 0,Y 437.557,Z 1101.07,A -85,B 0,C 180,E1 15896.038,E2 15896.038} C_VEL
LIN {X 0,Y 425.742,Z 1142.194,A -85,B 0,C 180,E1 15905.745,E2 15905.745} C_VEL
LIN {X 0,Y 420.147,Z 1168.326,A -85,B 0,C 180,E1 15915.834,E2 15915.834} C_VEL
LIN {X 0,Y 419.194,Z 1179.54,A -85,B 0,C 180,E1 15924.753,E2 15924.753} C_VEL
LIN {X 0,Y 419.261,Z 1180.587,A -85,B 0,C 180,E1 15933.057,E2 15933.057} C_VEL
LIN {X 0,Y 419.795,Z 1171.405,A -85,B 0,C 180,E1 15942.303,E2 15942.303} C_VEL
LIN {X 0,Y 424.001,Z 1149.058,A -85,B 0,C 180,E1 15952.012,E2 15952.012} C_VEL
LIN {X 0,Y 434.55,Z 1110.843,A -85,B 0,C 180,E1 15961.935,E2 15961.935} C_VEL
LIN {X 0,Y 450.91,Z 1059.03,A -85,B 0,C 180,E1 15970.623,E2 15970.623} C_VEL
LIN {X 0,Y 470.694,Z 995.915,A -85,B 0,C 180,E1 15977.579,E2 15977.579} C_VEL
LIN {X 0,Y 481.013,Z 958.176,A -85,B 0,C 180,E1 15980.534,E2 15980.534} C_VEL
LIN {X 0,Y 438.317,Z 989.946,A -85,B 0,C 180,E1 15983.544,E2 15983.544} C_VEL
LIN {X 0,Y 427.968,Z 994.752,A -85,B 0,C 180,E1 15984.897,E2 15984.897} C_VEL
LIN {X 0,Y 426.531,Z 1036.987,A -85,B 0,C 180,E1 15987.282,E2 15987.282} C_VEL
LIN {X 0,Y 424.248,Z 1069.805,A -85,B 0,C 180,E1 15991.2,E2 15991.2} C_VEL
LIN {X 0,Y 422.638,Z 1090.392,A -85,B 0,C 180,E1 15996.14,E2 15996.14} C_VEL
LIN {X 0,Y 422.303,Z 1096.943,A -85,B 0,C 180,E1 16000.107,E2 16000.107} C_VEL
LIN {X 0,Y 423.069,Z 1094.25,A -85,B 0,C 180,E1 16005.203,E2 16005.203} C_VEL
LIN {X 0,Y 425.137,Z 1076.798,A -85,B 0,C 180,E1 16010.389,E2 16010.389} C_VEL
LIN {X 0,Y 427.181,Z 1046.341,A -85,B 0,C 180,E1 16014.49,E2 16014.49} C_VEL
LIN {X 0,Y 428.537,Z 1006.318,A -85,B 0,C 180,E1 16017.015,E2 16017.015} C_VEL
LIN {X 0,Y 431.907,Z 869.745,A -85,B 0,C 180,E1 16020.237,E2 16020.237} C_VEL
LIN {X 0,Y 432.133,Z 814.478,A -85,B 0,C 180,E1 16022.952,E2 16022.952} C_VEL
LIN {X 0,Y 439.31,Z 791.168,A -85,B 0,C 180,E1 16026.072,E2 16026.072} C_VEL
LIN {X 0,Y 450.715,Z 807.295,A -85,B 0,C 180,E1 16034.756,E2 16034.756} C_VEL
LIN {X 0,Y 472.077,Z 841.756,A -85,B 0,C 180,E1 16044.186,E2 16044.186} C_VEL
LIN {X 0,Y 497.472,Z 889.463,A -85,B 0,C 180,E1 16052.319,E2 16052.319} C_VEL
LIN {X 0,Y 504.444,Z 908.701,A -85,B 0,C 180,E1 16054.621,E2 16054.621} C_VEL
LIN {X 0,Y 487.092,Z 990.203,A -85,B 0,C 180,E1 16058.65,E2 16058.65} C_VEL
LIN {X 0,Y 470.013,Z 1054.815,A -85,B 0,C 180,E1 16063.647,E2 16063.647} C_VEL
LIN {X 0,Y 451.457,Z 1109.263,A -85,B 0,C 180,E1 16070.334,E2 16070.334} C_VEL
LIN {X 0,Y 434.726,Z 1153.281,A -85,B 0,C 180,E1 16078.882,E2 16078.882} C_VEL
LIN {X 0,Y 423.572,Z 1185.508,A -85,B 0,C 180,E1 16089.289,E2 16089.289} C_VEL
LIN {X 0,Y 419.437,Z 1202.859,A -85,B 0,C 180,E1 16099.635,E2 16099.635} C_VEL
LIN {X 0,Y 419.503,Z 1208.69,A -85,B 0,C 180,E1 16109.019,E2 16109.019} C_VEL
LIN {X 0,Y 419.416,Z 1203.889,A -85,B 0,C 180,E1 16119.425,E2 16119.425} C_VEL
LIN {X 0,Y 422.91,Z 1187.152,A -85,B 0,C 180,E1 16129.986,E2 16129.986} C_VEL
LIN {X 0,Y 425.975,Z 1176.329,A -85,B 0,C 180,E1 16134.335,E2 16134.335} C_VEL
LIN {X 0,Y 423.333,Z 1163.609,A -85,B 0,C 180,E1 16138.811,E2 16138.811} C_VEL
LIN {X 0,Y 439.148,Z 1123.55,A -85,B 0,C 180,E1 16147.895,E2 16147.895} C_VEL
LIN {X 0,Y 458.282,Z 1072.095,A -85,B 0,C 180,E1 16155.208,E2 16155.208} C_VEL
LIN {X 0,Y 476.349,Z 1011.601,A -85,B 0,C 180,E1 16160.657,E2 16160.657} C_VEL
LIN {X 0,Y 495.736,Z 926.905,A -85,B 0,C 180,E1 16165.368,E2 16165.368} C_VEL
LIN {X 0,Y 498.201,Z 906.945,A -85,B 0,C 180,E1 16166.408,E2 16166.408} C_VEL
LIN {X 0,Y 474.565,Z 858.403,A -85,B 0,C 180,E1 16174.053,E2 16174.053} C_VEL
LIN {X 0,Y 454.426,Z 825.042,A -85,B 0,C 180,E1 16182.141,E2 16182.141} C_VEL
LIN {X 0,Y 441.075,Z 804.675,A -85,B 0,C 180,E1 16190.334,E2 16190.334} C_VEL
LIN {X 0,Y 435.097,Z 792.932,A -85,B 0,C 180,E1 16198.942,E2 16198.942} C_VEL
LIN {X 0,Y 435.318,Z 795.948,A -85,B 0,C 180,E1 16207.074,E2 16207.074} C_VEL
LIN {X 0,Y 443.422,Z 807.692,A -85,B 0,C 180,E1 16215.572,E2 16215.572} C_VEL
LIN {X 0,Y 459.991,Z 834.617,A -85,B 0,C 180,E1 16224.289,E2 16224.289} C_VEL
LIN {X 0,Y 480.368,Z 873.466,A -85,B 0,C 180,E1 16231.631,E2 16231.631} C_VEL
LIN {X 0,Y 488.294,Z 907.645,A -85,B 0,C 180,E1 16235.686,E2 16235.686} C_VEL
LIN {X 0,Y 469.467,Z 981.369,A -85,B 0,C 180,E1 16240.325,E2 16240.325} C_VEL
LIN {X 0,Y 448.932,Z 1046.368,A -85,B 0,C 180,E1 16246.905,E2 16246.905} C_VEL
LIN {X 0,Y 430.786,Z 1100.844,A -85,B 0,C 180,E1 16255.346,E2 16255.346} C_VEL
LIN {X 0,Y 418.223,Z 1142.285,A -85,B 0,C 180,E1 16265.28,E2 16265.28} C_VEL
LIN {X 0,Y 412.493,Z 1167.406,A -85,B 0,C 180,E1 16275.021,E2 16275.021} C_VEL
LIN {X 0,Y 411.194,Z 1179.77,A -85,B 0,C 180,E1 16284.65,E2 16284.65} C_VEL
LIN {X 0,Y 411.255,Z 1180.835,A -85,B 0,C 180,E1 16293.116,E2 16293.116} C_VEL
LIN {X 0,Y 411.961,Z 1171.038,A -85,B 0,C 180,E1 16302.861,E2 16302.861} C_VEL
LIN {X 0,Y 416.804,Z 1147.584,A -85,B 0,C 180,E1 16312.978,E2 16312.978} C_VEL
LIN {X 0,Y 428.14,Z 1108.853,A -85,B 0,C 180,E1 16322.953,E2 16322.953} C_VEL
LIN {X 0,Y 445.717,Z 1056.096,A -85,B 0,C 180,E1 16331.736,E2 16331.736} C_VEL
LIN {X 0,Y 465.999,Z 993.091,A -85,B 0,C 180,E1 16338.581,E2 16338.581} C_VEL
LIN {X 0,Y 471.312,Z 971.899,A -85,B 0,C 180,E1 16340.43,E2 16340.43} C_VEL
LIN {X 0,Y 431.628,Z 998.928,A -85,B 0,C 180,E1 16343.377,E2 16343.377} C_VEL
LIN {X 0,Y 419.982,Z 1004.863,A -85,B 0,C 180,E1 16345,E2 16345} C_VEL
LIN {X 0,Y 418.394,Z 1045.06,A -85,B 0,C 180,E1 16347.744,E2 16347.744} C_VEL
LIN {X 0,Y 416,Z 1076.228,A -85,B 0,C 180,E1 16352.062,E2 16352.062} C_VEL
LIN {X 0,Y 414.52,Z 1094.59,A -85,B 0,C 180,E1 16357.465,E2 16357.465} C_VEL
LIN {X 0,Y 414.654,Z 1098.093,A -85,B 0,C 180,E1 16363.043,E2 16363.043} C_VEL
LIN {X 0,Y 416.419,Z 1086.941,A -85,B 0,C 180,E1 16368.502,E2 16368.502} C_VEL
LIN {X 0,Y 418.608,Z 1061.786,A -85,B 0,C 180,E1 16373.186,E2 16373.186} C_VEL
LIN {X 0,Y 420.722,Z 1024.424,A -85,B 0,C 180,E1 16376.507,E2 16376.507} C_VEL
LIN {X 0,Y 421.06,Z 974.144,A -85,B 0,C 180,E1 16378.189,E2 16378.189} C_VEL
LIN {X 0,Y 424.516,Z 871.147,A -85,B 0,C 180,E1 16380.626,E2 16380.626} C_VEL
LIN {X 0,Y 427.403,Z 825.335,A -85,B 0,C 180,E1 16383.049,E2 16383.049} C_VEL
LIN {X 0,Y 437.712,Z 799.26,A -85,B 0,C 180,E1 16386.477,E2 16386.477} C_VEL
LIN {X 0,Y 448.582,Z 815.837,A -85,B 0,C 180,E1 16394.828,E2 16394.828} C_VEL
LIN {X 0,Y 468.431,Z 848.243,A -85,B 0,C 180,E1 16403.816,E2 16403.816} C_VEL
LIN {X 0,Y 492.962,Z 895.459,A -85,B 0,C 180,E1 16412.002,E2 16412.002} C_VEL
LIN {X 0,Y 498.749,Z 912.033,A -85,B 0,C 180,E1 16414.028,E2 16414.028} C_VEL
LIN {X 0,Y 480.625,Z 994.136,A -85,B 0,C 180,E1 16418.187,E2 16418.187} C_VEL
LIN {X 0,Y 463.096,Z 1057.37,A -85,B 0,C 180,E1 16423.226,E2 16423.226} C_VEL
LIN {X 0,Y 444.255,Z 1110.554,A -85,B 0,C 180,E1 16429.928,E2 16429.928} C_VEL
LIN {X 0,Y 427.005,Z 1154.281,A -85,B 0,C 180,E1 16438.653,E2 16438.653} C_VEL
LIN {X 0,Y 415.656,Z 1185.971,A -85,B 0,C 180,E1 16449.161,E2 16449.161} C_VEL
LIN {X 0,Y 411.484,Z 1202.744,A -85,B 0,C 180,E1 16459.432,E2 16459.432} C_VEL
LIN {X 0,Y 411.501,Z 1208.429,A -85,B 0,C 180,E1 16469,E2 16469} C_VEL
LIN {X 0,Y 411.447,Z 1203.76,A -85,B 0,C 180,E1 16479.609,E2 16479.609} C_VEL
LIN {X 0,Y 415.091,Z 1186.974,A -85,B 0,C 180,E1 16490.379,E2 16490.379} C_VEL
LIN {X 0,Y 423.333,Z 1163.609,A -85,B 0,C 180,E1 16498.811,E2 16498.811} C_VEL
LIN {X 0,Y 421.512,Z 1148.973,A -85,B 0,C 180,E1 16503.193,E2 16503.193} C_VEL
LIN {X 0,Y 439.866,Z 1104.292,A -85,B 0,C 180,E1 16511.679,E2 16511.679} C_VEL
LIN {X 0,Y 460.205,Z 1047.915,A -85,B 0,C 180,E1 16518.394,E2 16518.394} C_VEL
LIN {X 0,Y 478.216,Z 981.616,A -85,B 0,C 180,E1 16523.331,E2 16523.331} C_VEL
LIN {X 0,Y 493.122,Z 911.957,A -85,B 0,C 180,E1 16526.838,E2 16526.838} C_VEL
LIN {X 0,Y 470.262,Z 863.91,A -85,B 0,C 180,E1 16534.567,E2 16534.567} C_VEL
LIN {X 0,Y 450.313,Z 830.014,A -85,B 0,C 180,E1 16543.063,E2 16543.063} C_VEL
LIN {X 0,Y 436.737,Z 807.739,A -85,B 0,C 180,E1 16552.681,E2 16552.681} C_VEL
LIN {X 0,Y 432.519,Z 800.604,A -85,B 0,C 180,E1 16560.946,E2 16560.946} C_VEL
LIN {X 0,Y 433.686,Z 804.764,A -85,B 0,C 180,E1 16567.985,E2 16567.985} C_VEL
LIN {X 0,Y 441.165,Z 815.774,A -85,B 0,C 180,E1 16575.526,E2 16575.526} C_VEL
LIN {X 0,Y 456.989,Z 841.637,A -85,B 0,C 180,E1 16583.989,E2 16583.989} C_VEL
LIN {X 0,Y 475.977,Z 879.031,A -85,B 0,C 180,E1 16591.183,E2 16591.183} C_VEL
LIN {X 0,Y 482.849,Z 911.1,A -85,B 0,C 180,E1 16595.083,E2 16595.083} C_VEL
LIN {X 0,Y 463.401,Z 984.167,A -85,B 0,C 180,E1 16599.766,E2 16599.766} C_VEL
LIN {X 0,Y 441.537,Z 1050.404,A -85,B 0,C 180,E1 16606.658,E2 16606.658} C_VEL
LIN {X 0,Y 423.456,Z 1102.346,A -85,B 0,C 180,E1 16614.975,E2 16614.975} C_VEL
LIN {X 0,Y 410.74,Z 1142.425,A -85,B 0,C 180,E1 16624.798,E2 16624.798} C_VEL
LIN {X 0,Y 404.64,Z 1167.572,A -85,B 0,C 180,E1 16634.723,E2 16634.723} C_VEL
LIN {X 0,Y 403.191,Z 1180.004,A -85,B 0,C 180,E1 16644.544,E2 16644.544} C_VEL
LIN {X 0,Y 403.248,Z 1181.085,A -85,B 0,C 180,E1 16653.178,E2 16653.178} C_VEL
LIN {X 0,Y 404.046,Z 1171.224,A -85,B 0,C 180,E1 16663.117,E2 16663.117} C_VEL
LIN {X 0,Y 409.19,Z 1147.741,A -85,B 0,C 180,E1 16673.431,E2 16673.431} C_VEL
LIN {X 0,Y 421.12,Z 1108.996,A -85,B 0,C 180,E1 16683.574,E2 16683.574} C_VEL
LIN {X 0,Y 439.112,Z 1057.483,A -85,B 0,C 180,E1 16692.291,E2 16692.291} C_VEL
LIN {X 0,Y 460.065,Z 994.943,A -85,B 0,C 180,E1 16699.202,E2 16699.202} C_VEL
LIN {X 0,Y 462.268,Z 984.379,A -85,B 0,C 180,E1 16700.278,E2 16700.278} C_VEL
LIN {X 0,Y 424.982,Z 1007.188,A -85,B 0,C 180,E1 16703.285,E2 16703.285} C_VEL
LIN {X 0,Y 411.983,Z 1013.084,A -85,B 0,C 180,E1 16705.106,E2 16705.106} C_VEL
LIN {X 0,Y 410.015,Z 1053.271,A -85,B 0,C 180,E1 16708.33,E2 16708.33} C_VEL
LIN {X 0,Y 407.876,Z 1081.567,A -85,B 0,C 180,E1 16712.866,E2 16712.866} C_VEL
LIN {X 0,Y 406.519,Z 1097.349,A -85,B 0,C 180,E1 16718.424,E2 16718.424} C_VEL
LIN {X 0,Y 406.931,Z 1098.69,A -85,B 0,C 180,E1 16723.827,E2 16723.827} C_VEL
LIN {X 0,Y 408.873,Z 1085.959,A -85,B 0,C 180,E1 16729.246,E2 16729.246} C_VEL
LIN {X 0,Y 411.189,Z 1058.982,A -85,B 0,C 180,E1 16733.923,E2 16733.923} C_VEL
LIN {X 0,Y 413.274,Z 1020.552,A -85,B 0,C 180,E1 16737.102,E2 16737.102} C_VEL
LIN {X 0,Y 413.804,Z 953.636,A -85,B 0,C 180,E1 16739.011,E2 16739.011} C_VEL
LIN {X 0,Y 417.313,Z 870.876,A -85,B 0,C 180,E1 16741.103,E2 16741.103} C_VEL
LIN {X 0,Y 419.714,Z 850.379,A -85,B 0,C 180,E1 16742.392,E2 16742.392} C_VEL
LIN {X 0,Y 429.773,Z 822.094,A -85,B 0,C 180,E1 16744.806,E2 16744.806} C_VEL
LIN {X 0,Y 436.271,Z 807.494,A -85,B 0,C 180,E1 16747.05,E2 16747.05} C_VEL
LIN {X 0,Y 447.905,Z 826.458,A -85,B 0,C 180,E1 16755.747,E2 16755.747} C_VEL
LIN {X 0,Y 467.684,Z 859.929,A -85,B 0,C 180,E1 16764.557,E2 16764.557} C_VEL
LIN {X 0,Y 490.875,Z 907.056,A -85,B 0,C 180,E1 16772.48,E2 16772.48} C_VEL
LIN {X 0,Y 492.806,Z 917.221,A -85,B 0,C 180,E1 16773.504,E2 16773.504} C_VEL
LIN {X 0,Y 473.968,Z 999.367,A -85,B 0,C 180,E1 16777.79,E2 16777.79} C_VEL
LIN {X 0,Y 455.33,Z 1062.43,A -85,B 0,C 180,E1 16783.051,E2 16783.051} C_VEL
LIN {X 0,Y 435.879,Z 1114.674,A -85,B 0,C 180,E1 16789.978,E2 16789.978} C_VEL
LIN {X 0,Y 418.478,Z 1157.307,A -85,B 0,C 180,E1 16798.954,E2 16798.954} C_VEL
LIN {X 0,Y 407.046,Z 1188.143,A -85,B 0,C 180,E1 16809.89,E2 16809.89} C_VEL
LIN {X 0,Y 403.356,Z 1203.675,A -85,B 0,C 180,E1 16820.312,E2 16820.312} C_VEL
LIN {X 0,Y 403.493,Z 1208.168,A -85,B 0,C 180,E1 16828.98,E2 16828.98} C_VEL
LIN {X 0,Y 403.48,Z 1203.572,A -85,B 0,C 180,E1 16839.801,E2 16839.801} C_VEL
LIN {X 0,Y 407.292,Z 1186.725,A -85,B 0,C 180,E1 16850.788,E2 16850.788} C_VEL
LIN {X 0,Y 418.017,Z 1157.503,A -85,B 0,C 180,E1 16861.021,E2 16861.021} C_VEL
LIN {X 0,Y 421.512,Z 1148.973,A -85,B 0,C 180,E1 16863.193,E2 16863.193} C_VEL
LIN {X 0,Y 421.823,Z 1132.096,A -85,B 0,C 180,E1 16867.444,E2 16867.444} C_VEL
LIN {X 0,Y 441.823,Z 1082.922,A -85,B 0,C 180,E1 16875.275,E2 16875.275} C_VEL
LIN {X 0,Y 461.937,Z 1023.473,A -85,B 0,C 180,E1 16881.237,E2 16881.237} C_VEL
LIN {X 0,Y 481.799,Z 945.091,A -85,B 0,C 180,E1 16886.004,E2 16886.004} C_VEL
LIN {X 0,Y 487.441,Z 915.478,A -85,B 0,C 180,E1 16887.463,E2 16887.463} C_VEL
LIN {X 0,Y 465.331,Z 868.249,A -85,B 0,C 180,E1 16895.343,E2 16895.343} C_VEL
LIN {X 0,Y 445.717,Z 834.304,A -85,B 0,C 180,E1 16904.265,E2 16904.265} C_VEL
LIN {X 0,Y 433.903,Z 814.968,A -85,B 0,C 180,E1 16913.415,E2 16913.415} C_VEL
LIN {X 0,Y 430.492,Z 808.338,A -85,B 0,C 180,E1 16920.951,E2 16920.951} C_VEL
LIN {X 0,Y 431.598,Z 812.464,A -85,B 0,C 180,E1 16927.897,E2 16927.897} C_VEL
LIN {X 0,Y 438.868,Z 823.546,A -85,B 0,C 180,E1 16935.417,E2 16935.417} C_VEL
LIN {X 0,Y 454.061,Z 848.897,A -85,B 0,C 180,E1 16943.745,E2 16943.745} C_VEL
LIN {X 0,Y 472.075,Z 886.11,A -85,B 0,C 180,E1 16950.98,E2 16950.98} C_VEL
LIN {X 0,Y 477.215,Z 915.517,A -85,B 0,C 180,E1 16954.509,E2 16954.509} C_VEL
LIN {X 0,Y 457.319,Z 987,A -85,B 0,C 180,E1 16959.199,E2 16959.199} C_VEL
LIN {X 0,Y 434.66,Z 1053,A -85,B 0,C 180,E1 16966.218,E2 16966.218} C_VEL
LIN {X 0,Y 415.573,Z 1105.332,A -85,B 0,C 180,E1 16974.893,E2 16974.893} C_VEL
LIN {X 0,Y 402.108,Z 1146.123,A -85,B 0,C 180,E1 16985.413,E2 16985.413} C_VEL
LIN {X 0,Y 396.314,Z 1169.755,A -85,B 0,C 180,E1 16995.53,E2 16995.53} C_VEL
LIN {X 0,Y 395.191,Z 1180.25,A -85,B 0,C 180,E1 17004.433,E2 17004.433} C_VEL
LIN {X 0,Y 395.254,Z 1181.34,A -85,B 0,C 180,E1 17013.243,E2 17013.243} C_VEL
LIN {X 0,Y 396.121,Z 1171.526,A -85,B 0,C 180,E1 17023.324,E2 17023.324} C_VEL
LIN {X 0,Y 401.621,Z 1147.932,A -85,B 0,C 180,E1 17033.9,E2 17033.9} C_VEL
LIN {X 0,Y 414.192,Z 1109.166,A -85,B 0,C 180,E1 17044.213,E2 17044.213} C_VEL
LIN {X 0,Y 433.592,Z 1056.124,A -85,B 0,C 180,E1 17053.255,E2 17053.255} C_VEL
LIN {X 0,Y 454.099,Z 995.421,A -85,B 0,C 180,E1 17060.043,E2 17060.043} C_VEL
LIN {X 0,Y 422.097,Z 1013.668,A -85,B 0,C 180,E1 17062.687,E2 17062.687} C_VEL
LIN {X 0,Y 404.014,Z 1021.375,A -85,B 0,C 180,E1 17065.277,E2 17065.277} C_VEL
LIN {X 0,Y 401.623,Z 1059.965,A -85,B 0,C 180,E1 17068.838,E2 17068.838} C_VEL
LIN {X 0,Y 399.592,Z 1087.062,A -85,B 0,C 180,E1 17073.867,E2 17073.867} C_VEL
LIN {X 0,Y 398.577,Z 1099.034,A -85,B 0,C 180,E1 17078.868,E2 17078.868} C_VEL
LIN {X 0,Y 399.208,Z 1099.143,A -85,B 0,C 180,E1 17084.549,E2 17084.549} C_VEL
LIN {X 0,Y 401.388,Z 1085.152,A -85,B 0,C 180,E1 17089.964,E2 17089.964} C_VEL
LIN {X 0,Y 403.777,Z 1057.687,A -85,B 0,C 180,E1 17094.511,E2 17094.511} C_VEL
LIN {X 0,Y 405.753,Z 1018.039,A -85,B 0,C 180,E1 17097.652,E2 17097.652} C_VEL
LIN {X 0,Y 409.644,Z 880.763,A -85,B 0,C 180,E1 17101.272,E2 17101.272} C_VEL
LIN {X 0,Y 428.891,Z 827.83,A -85,B 0,C 180,E1 17105.549,E2 17105.549} C_VEL
LIN {X 0,Y 434.596,Z 815.635,A -85,B 0,C 180,E1 17107.452,E2 17107.452} C_VEL
LIN {X 0,Y 448.155,Z 838.756,A -85,B 0,C 180,E1 17117.164,E2 17117.164} C_VEL
LIN {X 0,Y 467.89,Z 873.773,A -85,B 0,C 180,E1 17125.717,E2 17125.717} C_VEL
LIN {X 0,Y 487.831,Z 917.652,A -85,B 0,C 180,E1 17132.773,E2 17132.773} C_VEL
LIN {X 0,Y 468.423,Z 1000.007,A -85,B 0,C 180,E1 17137.087,E2 17137.087} C_VEL
LIN {X 0,Y 449.513,Z 1061.89,A -85,B 0,C 180,E1 17142.296,E2 17142.296} C_VEL
LIN {X 0,Y 429.435,Z 1114.068,A -85,B 0,C 180,E1 17149.252,E2 17149.252} C_VEL
LIN {X 0,Y 411.257,Z 1156.979,A -85,B 0,C 180,E1 17158.368,E2 17158.368} C_VEL
LIN {X 0,Y 399.314,Z 1187.876,A -85,B 0,C 180,E1 17169.483,E2 17169.483} C_VEL
LIN {X 0,Y 395.375,Z 1203.428,A -85,B 0,C 180,E1 17180.115,E2 17180.115} C_VEL
LIN {X 0,Y 395.5,Z 1207.906,A -85,B 0,C 180,E1 17188.959,E2 17188.959} C_VEL
LIN {X 0,Y 395.509,Z 1203.332,A -85,B 0,C 180,E1 17200,E2 17200} C_VEL
LIN {X 0,Y 399.598,Z 1186.147,A -85,B 0,C 180,E1 17211.352,E2 17211.352} C_VEL
LIN {X 0,Y 411.361,Z 1155.796,A -85,B 0,C 180,E1 17221.972,E2 17221.972} C_VEL
LIN {X 0,Y 421.823,Z 1132.096,A -85,B 0,C 180,E1 17227.444,E2 17227.444} C_VEL
LIN {X 0,Y 422.963,Z 1113.329,A -85,B 0,C 180,E1 17231.533,E2 17231.533} C_VEL
LIN {X 0,Y 444.157,Z 1060.153,A -85,B 0,C 180,E1 17238.618,E2 17238.618} C_VEL
LIN {X 0,Y 463.713,Z 997.032,A -85,B 0,C 180,E1 17243.911,E2 17243.911} C_VEL
LIN {X 0,Y 481.997,Z 919.529,A -85,B 0,C 180,E1 17248.04,E2 17248.04} C_VEL
LIN {X 0,Y 460.947,Z 873.687,A -85,B 0,C 180,E1 17255.902,E2 17255.902} C_VEL
LIN {X 0,Y 442.309,Z 840.789,A -85,B 0,C 180,E1 17264.841,E2 17264.841} C_VEL
LIN {X 0,Y 431.523,Z 822.515,A -85,B 0,C 180,E1 17273.632,E2 17273.632} C_VEL
LIN {X 0,Y 428.418,Z 816.065,A -85,B 0,C 180,E1 17280.955,E2 17280.955} C_VEL
LIN {X 0,Y 429.555,Z 820.416,A -85,B 0,C 180,E1 17288.062,E2 17288.062} C_VEL
LIN {X 0,Y 436.735,Z 831.777,A -85,B 0,C 180,E1 17295.494,E2 17295.494} C_VEL
LIN {X 0,Y 451.496,Z 856.771,A -85,B 0,C 180,E1 17303.655,E2 17303.655} C_VEL
LIN {X 0,Y 467.888,Z 892.475,A -85,B 0,C 180,E1 17310.656,E2 17310.656} C_VEL
LIN {X 0,Y 471.62,Z 920.068,A -85,B 0,C 180,E1 17313.931,E2 17313.931} C_VEL
LIN {X 0,Y 451.17,Z 990.174,A -85,B 0,C 180,E1 17318.647,E2 17318.647} C_VEL
LIN {X 0,Y 427.981,Z 1055.172,A -85,B 0,C 180,E1 17325.709,E2 17325.709} C_VEL
LIN {X 0,Y 407.85,Z 1107.891,A -85,B 0,C 180,E1 17334.715,E2 17334.715} C_VEL
LIN {X 0,Y 394.366,Z 1147.077,A -85,B 0,C 180,E1 17345.162,E2 17345.162} C_VEL
LIN {X 0,Y 388.44,Z 1169.969,A -85,B 0,C 180,E1 17355.23,E2 17355.23} C_VEL
LIN {X 0,Y 387.191,Z 1180.5,A -85,B 0,C 180,E1 17364.318,E2 17364.318} C_VEL
LIN {X 0,Y 387.226,Z 1181.452,A -85,B 0,C 180,E1 17373.62,E2 17373.62} C_VEL
LIN {X 0,Y 388.19,Z 1171.897,A -85,B 0,C 180,E1 17383.502,E2 17383.502} C_VEL
LIN {X 0,Y 393.971,Z 1148.427,A -85,B 0,C 180,E1 17394.284,E2 17394.284} C_VEL
LIN {X 0,Y 407.269,Z 1109.366,A -85,B 0,C 180,E1 17404.878,E2 17404.878} C_VEL
LIN {X 0,Y 427.494,Z 1056.579,A -85,B 0,C 180,E1 17413.99,E2 17413.99} C_VEL
LIN {X 0,Y 445.408,Z 1006.391,A -85,B 0,C 180,E1 17419.823,E2 17419.823} C_VEL
LIN {X 0,Y 407.438,Z 1024.728,A -85,B 0,C 180,E1 17423.507,E2 17423.507} C_VEL
LIN {X 0,Y 395.877,Z 1029.154,A -85,B 0,C 180,E1 17425.499,E2 17425.499} C_VEL
LIN {X 0,Y 393.301,Z 1066.194,A -85,B 0,C 180,E1 17429.388,E2 17429.388} C_VEL
LIN {X 0,Y 391.305,Z 1091.209,A -85,B 0,C 180,E1 17434.689,E2 17434.689} C_VEL
LIN {X 0,Y 390.678,Z 1101.016,A -85,B 0,C 180,E1 17439.611,E2 17439.611} C_VEL
LIN {X 0,Y 391.571,Z 1099.164,A -85,B 0,C 180,E1 17445.48,E2 17445.48} C_VEL
LIN {X 0,Y 393.977,Z 1083.048,A -85,B 0,C 180,E1 17450.925,E2 17450.925} C_VEL
LIN {X 0,Y 396.536,Z 1053.155,A -85,B 0,C 180,E1 17455.445,E2 17455.445} C_VEL
LIN {X 0,Y 398.377,Z 1012.968,A -85,B 0,C 180,E1 17458.291,E2 17458.291} C_VEL
LIN {X 0,Y 401.786,Z 904.345,A -85,B 0,C 180,E1 17461.245,E2 17461.245} C_VEL
LIN {X 0,Y 416.751,Z 863.18,A -85,B 0,C 180,E1 17463.773,E2 17463.773} C_VEL
LIN {X 0,Y 429.394,Z 830.763,A -85,B 0,C 180,E1 17466.718,E2 17466.718} C_VEL
LIN {X 0,Y 432.612,Z 824.507,A -85,B 0,C 180,E1 17467.807,E2 17467.807} C_VEL
LIN {X 0,Y 445.178,Z 845.905,A -85,B 0,C 180,E1 17476.9,E2 17476.9} C_VEL
LIN {X 0,Y 464.538,Z 881.446,A -85,B 0,C 180,E1 17485.609,E2 17485.609} C_VEL
LIN {X 0,Y 482.299,Z 920.956,A -85,B 0,C 180,E1 17492.138,E2 17492.138} C_VEL
LIN {X 0,Y 461.794,Z 1004.785,A -85,B 0,C 180,E1 17496.645,E2 17496.645} C_VEL
LIN {X 0,Y 441.559,Z 1067.256,A -85,B 0,C 180,E1 17502.148,E2 17502.148} C_VEL
LIN {X 0,Y 420.028,Z 1120.194,A -85,B 0,C 180,E1 17509.664,E2 17509.664} C_VEL
LIN {X 0,Y 402.119,Z 1160.904,A -85,B 0,C 180,E1 17518.991,E2 17518.991} C_VEL
LIN {X 0,Y 390.728,Z 1189.778,A -85,B 0,C 180,E1 17530.199,E2 17530.199} C_VEL
LIN {X 0,Y 387.4,Z 1203.165,A -85,B 0,C 180,E1 17539.909,E2 17539.909} C_VEL
LIN {X 0,Y 387.355,Z 1207.694,A -85,B 0,C 180,E1 17549.556,E2 17549.556} C_VEL
LIN {X 0,Y 387.524,Z 1203.068,A -85,B 0,C 180,E1 17560.209,E2 17560.209} C_VEL
LIN {X 0,Y 391.764,Z 1186.135,A -85,B 0,C 180,E1 17571.652,E2 17571.652} C_VEL
LIN {X 0,Y 404.04,Z 1155.926,A -85,B 0,C 180,E1 17582.455,E2 17582.455} C_VEL
LIN {X 0,Y 422.963,Z 1113.329,A -85,B 0,C 180,E1 17591.533,E2 17591.533} C_VEL
LIN {X 0,Y 425.444,Z 1092.531,A -85,B 0,C 180,E1 17595.405,E2 17595.405} C_VEL
LIN {X 0,Y 447.129,Z 1035.123,A -85,B 0,C 180,E1 17601.78,E2 17601.78} C_VEL
LIN {X 0,Y 466.422,Z 967.711,A -85,B 0,C 180,E1 17606.393,E2 17606.393} C_VEL
LIN {X 0,Y 476.029,Z 922.217,A -85,B 0,C 180,E1 17608.818,E2 17608.818} C_VEL
LIN {X 0,Y 455.192,Z 876.08,A -85,B 0,C 180,E1 17617.117,E2 17617.117} C_VEL
LIN {X 0,Y 436.959,Z 843.305,A -85,B 0,C 180,E1 17626.768,E2 17626.768} C_VEL
LIN {X 0,Y 428.178,Z 829.225,A -85,B 0,C 180,E1 17634.985,E2 17634.985} C_VEL
LIN {X 0,Y 426.296,Z 823.778,A -85,B 0,C 180,E1 17640.96,E2 17640.96} C_VEL
LIN {X 0,Y 427.42,Z 828.107,A -85,B 0,C 180,E1 17647.974,E2 17647.974} C_VEL
LIN {X 0,Y 434.302,Z 839.344,A -85,B 0,C 180,E1 17655.324,E2 17655.324} C_VEL
LIN {X 0,Y 448.947,Z 864.678,A -85,B 0,C 180,E1 17663.599,E2 17663.599} C_VEL
LIN {X 0,Y 464.251,Z 900.809,A -85,B 0,C 180,E1 17670.647,E2 17670.647} C_VEL
LIN {X 0,Y 466.061,Z 924.533,A -85,B 0,C 180,E1 17673.333,E2 17673.333} C_VEL
LIN {X 0,Y 444.511,Z 994.994,A -85,B 0,C 180,E1 17678.233,E2 17678.233} C_VEL
LIN {X 0,Y 421.068,Z 1057.971,A -85,B 0,C 180,E1 17685.28,E2 17685.28} C_VEL
LIN {X 0,Y 399.883,Z 1111.098,A -85,B 0,C 180,E1 17694.671,E2 17694.671} C_VEL
LIN {X 0,Y 385.917,Z 1149.839,A -85,B 0,C 180,E1 17705.551,E2 17705.551} C_VEL
LIN {X 0,Y 380.185,Z 1172.102,A -85,B 0,C 180,E1 17716.083,E2 17716.083} C_VEL
LIN {X 0,Y 379.194,Z 1181.846,A -85,B 0,C 180,E1 17726.498,E2 17726.498} C_VEL
LIN {X 0,Y 379.246,Z 1180.774,A -85,B 0,C 180,E1 17735.679,E2 17735.679} C_VEL
LIN {X 0,Y 381.461,Z 1167.296,A -85,B 0,C 180,E1 17746.698,E2 17746.698} C_VEL
LIN {X 0,Y 389.057,Z 1139.52,A -85,B 0,C 180,E1 17757.838,E2 17757.838} C_VEL
LIN {X 0,Y 405.42,Z 1096.295,A -85,B 0,C 180,E1 17768.332,E2 17768.332} C_VEL
LIN {X 0,Y 427.694,Z 1040.91,A -85,B 0,C 180,E1 17776.858,E2 17776.858} C_VEL
LIN {X 0,Y 436.588,Z 1016.547,A -85,B 0,C 180,E1 17779.668,E2 17779.668} C_VEL
LIN {X 0,Y 397.651,Z 1032.967,A -85,B 0,C 180,E1 17783.823,E2 17783.823} C_VEL
LIN {X 0,Y 387.784,Z 1036.709,A -85,B 0,C 180,E1 17785.78,E2 17785.78} C_VEL
LIN {X 0,Y 385.053,Z 1072.303,A -85,B 0,C 180,E1 17790.055,E2 17790.055} C_VEL
LIN {X 0,Y 383.132,Z 1094.756,A -85,B 0,C 180,E1 17795.503,E2 17795.503} C_VEL
LIN {X 0,Y 382.756,Z 1102.617,A -85,B 0,C 180,E1 17800.38,E2 17800.38} C_VEL
LIN {X 0,Y 383.946,Z 1098.838,A -85,B 0,C 180,E1 17806.482,E2 17806.482} C_VEL
LIN {X 0,Y 386.649,Z 1081.002,A -85,B 0,C 180,E1 17811.889,E2 17811.889} C_VEL
LIN {X 0,Y 389.303,Z 1050.345,A -85,B 0,C 180,E1 17816.199,E2 17816.199} C_VEL
LIN {X 0,Y 391.024,Z 1009.749,A -85,B 0,C 180,E1 17818.884,E2 17818.884} C_VEL
LIN {X 0,Y 393.584,Z 927.247,A -85,B 0,C 180,E1 17821.169,E2 17821.169} C_VEL
LIN {X 0,Y 413.168,Z 875.498,A -85,B 0,C 180,E1 17824.225,E2 17824.225} C_VEL
LIN {X 0,Y 428.208,Z 837.471,A -85,B 0,C 180,E1 17827.312,E2 17827.312} C_VEL
LIN {X 0,Y 430.75,Z 833.436,A -85,B 0,C 180,E1 17828.287,E2 17828.287} C_VEL
LIN {X 0,Y 443.78,Z 855.385,A -85,B 0,C 180,E1 17837.467,E2 17837.467} C_VEL
LIN {X 0,Y 463.167,Z 893.204,A -85,B 0,C 180,E1 17846.308,E2 17846.308} C_VEL
LIN {X 0,Y 476.293,Z 926.504,A -85,B 0,C 180,E1 17851.588,E2 17851.588} C_VEL
LIN {X 0,Y 455.308,Z 1009.093,A -85,B 0,C 180,E1 17856.171,E2 17856.171} C_VEL
LIN {X 0,Y 434.329,Z 1070.371,A -85,B 0,C 180,E1 17861.771,E2 17861.771} C_VEL
LIN {X 0,Y 412.536,Z 1121.893,A -85,B 0,C 180,E1 17869.326,E2 17869.326} C_VEL
LIN {X 0,Y 394.306,Z 1161.872,A -85,B 0,C 180,E1 17878.77,E2 17878.77} C_VEL
LIN {X 0,Y 382.565,Z 1190.534,A -85,B 0,C 180,E1 17890.362,E2 17890.362} C_VEL
LIN {X 0,Y 379.436,Z 1202.894,A -85,B 0,C 180,E1 17899.695,E2 17899.695} C_VEL
LIN {X 0,Y 379.523,Z 1207.381,A -85,B 0,C 180,E1 17908.915,E2 17908.915} C_VEL
LIN {X 0,Y 379.547,Z 1202.796,A -85,B 0,C 180,E1 17920.426,E2 17920.426} C_VEL
LIN {X 0,Y 384.014,Z 1185.805,A -85,B 0,C 180,E1 17932.112,E2 17932.112} C_VEL
LIN {X 0,Y 396.315,Z 1156.818,A -85,B 0,C 180,E1 17942.722,E2 17942.722} C_VEL
LIN {X 0,Y 415.992,Z 1114.21,A -85,B 0,C 180,E1 17952.055,E2 17952.055} C_VEL
LIN {X 0,Y 425.444,Z 1092.531,A -85,B 0,C 180,E1 17955.405,E2 17955.405} C_VEL
LIN {X 0,Y 428.718,Z 1069.806,A -85,B 0,C 180,E1 17959.047,E2 17959.047} C_VEL
LIN {X 0,Y 450.101,Z 1008.717,A -85,B 0,C 180,E1 17964.674,E2 17964.674} C_VEL
LIN {X 0,Y 470.639,Z 926.265,A -85,B 0,C 180,E1 17969.423,E2 17969.423} C_VEL
LIN {X 0,Y 450.819,Z 881.513,A -85,B 0,C 180,E1 17977.723,E2 17977.723} C_VEL
LIN {X 0,Y 433.817,Z 850.159,A -85,B 0,C 180,E1 17987.249,E2 17987.249} C_VEL
LIN {X 0,Y 425.855,Z 836.818,A -85,B 0,C 180,E1 17995.086,E2 17995.086} C_VEL
LIN {X 0,Y 424.158,Z 831.466,A -85,B 0,C 180,E1 18000.965,E2 18000.965} C_VEL
LIN {X 0,Y 425.235,Z 835.901,A -85,B 0,C 180,E1 18008.016,E2 18008.016} C_VEL
LIN {X 0,Y 432.114,Z 847.525,A -85,B 0,C 180,E1 18015.403,E2 18015.403} C_VEL
LIN {X 0,Y 446.42,Z 872.797,A -85,B 0,C 180,E1 18023.605,E2 18023.605} C_VEL
LIN {X 0,Y 460.426,Z 909.123,A -85,B 0,C 180,E1 18030.651,E2 18030.651} C_VEL
LIN {X 0,Y 460.753,Z 928.049,A -85,B 0,C 180,E1 18032.665,E2 18032.665} C_VEL
LIN {X 0,Y 438.611,Z 997.796,A -85,B 0,C 180,E1 18037.623,E2 18037.623} C_VEL
LIN {X 0,Y 414.583,Z 1059.696,A -85,B 0,C 180,E1 18044.682,E2 18044.682} C_VEL
LIN {X 0,Y 393.143,Z 1111.332,A -85,B 0,C 180,E1 18053.972,E2 18053.972} C_VEL
LIN {X 0,Y 378.47,Z 1150.079,A -85,B 0,C 180,E1 18065.038,E2 18065.038} C_VEL
LIN {X 0,Y 372.309,Z 1172.351,A -85,B 0,C 180,E1 18075.782,E2 18075.782} C_VEL
LIN {X 0,Y 371.198,Z 1182.105,A -85,B 0,C 180,E1 18086.422,E2 18086.422} C_VEL
LIN {X 0,Y 371.261,Z 1181.03,A -85,B 0,C 180,E1 18095.802,E2 18095.802} C_VEL
LIN {X 0,Y 373.568,Z 1167.545,A -85,B 0,C 180,E1 18107.061,E2 18107.061} C_VEL
LIN {X 0,Y 381.704,Z 1139.747,A -85,B 0,C 180,E1 18118.422,E2 18118.422} C_VEL
LIN {X 0,Y 398.437,Z 1097.67,A -85,B 0,C 180,E1 18128.855,E2 18128.855} C_VEL
LIN {X 0,Y 421.454,Z 1042.759,A -85,B 0,C 180,E1 18137.484,E2 18137.484} C_VEL
LIN {X 0,Y 427.932,Z 1025.86,A -85,B 0,C 180,E1 18139.502,E2 18139.502} C_VEL
LIN {X 0,Y 393.453,Z 1039.139,A -85,B 0,C 180,E1 18143.374,E2 18143.374} C_VEL
LIN {X 0,Y 379.669,Z 1043.552,A -85,B 0,C 180,E1 18146.068,E2 18146.068} C_VEL
LIN {X 0,Y 376.972,Z 1076.918,A -85,B 0,C 180,E1 18150.537,E2 18150.537} C_VEL
LIN {X 0,Y 375.07,Z 1098.198,A -85,B 0,C 180,E1 18156.402,E2 18156.402} C_VEL
LIN {X 0,Y 375.069,Z 1104.217,A -85,B 0,C 180,E1 18162.41,E2 18162.41} C_VEL
LIN {X 0,Y 377.013,Z 1095.543,A -85,B 0,C 180,E1 18168.578,E2 18168.578} C_VEL
LIN {X 0,Y 379.833,Z 1073.36,A -85,B 0,C 180,E1 18173.761,E2 18173.761} C_VEL
LIN {X 0,Y 382.651,Z 1039.177,A -85,B 0,C 180,E1 18177.652,E2 18177.652} C_VEL
LIN {X 0,Y 383.7,Z 995.582,A -85,B 0,C 180,E1 18179.783,E2 18179.783} C_VEL
LIN {X 0,Y 385.539,Z 946.794,A -85,B 0,C 180,E1 18181.194,E2 18181.194} C_VEL
LIN {X 0,Y 414.419,Z 875.095,A -85,B 0,C 180,E1 18185.471,E2 18185.471} C_VEL
LIN {X 0,Y 428.056,Z 842.129,A -85,B 0,C 180,E1 18188.211,E2 18188.211} C_VEL
LIN {X 0,Y 435.624,Z 853.803,A -85,B 0,C 180,E1 18194.16,E2 18194.16} C_VEL
LIN {X 0,Y 452.389,Z 885.304,A -85,B 0,C 180,E1 18203.074,E2 18203.074} C_VEL
LIN {X 0,Y 471.108,Z 928.167,A -85,B 0,C 180,E1 18210.838,E2 18210.838} C_VEL
LIN {X 0,Y 449.848,Z 1009.83,A -85,B 0,C 180,E1 18215.43,E2 18215.43} C_VEL
LIN {X 0,Y 428.452,Z 1070.281,A -85,B 0,C 180,E1 18221.008,E2 18221.008} C_VEL
LIN {X 0,Y 405.478,Z 1122.752,A -85,B 0,C 180,E1 18228.816,E2 18228.816} C_VEL
LIN {X 0,Y 386.24,Z 1163.233,A -85,B 0,C 180,E1 18238.703,E2 18238.703} C_VEL
LIN {X 0,Y 374.412,Z 1191.27,A -85,B 0,C 180,E1 18250.533,E2 18250.533} C_VEL
LIN {X 0,Y 371.303,Z 1204.44,A -85,B 0,C 180,E1 18261.84,E2 18261.84} C_VEL
LIN {X 0,Y 371.142,Z 1207.094,A -85,B 0,C 180,E1 18271.233,E2 18271.233} C_VEL
LIN {X 0,Y 371.737,Z 1201.538,A -85,B 0,C 180,E1 18281.68,E2 18281.68} C_VEL
LIN {X 0,Y 376.768,Z 1184.251,A -85,B 0,C 180,E1 18293.186,E2 18293.186} C_VEL
LIN {X 0,Y 390.1,Z 1154.674,A -85,B 0,C 180,E1 18303.876,E2 18303.876} C_VEL
LIN {X 0,Y 410.598,Z 1111.513,A -85,B 0,C 180,E1 18313.207,E2 18313.207} C_VEL
LIN {X 0,Y 428.718,Z 1069.806,A -85,B 0,C 180,E1 18319.047,E2 18319.047} C_VEL
LIN {X 0,Y 432.562,Z 1045.262,A -85,B 0,C 180,E1 18322.427,E2 18322.427} C_VEL
LIN {X 0,Y 452.852,Z 981.769,A -85,B 0,C 180,E1 18327.236,E2 18327.236} C_VEL
LIN {X 0,Y 465.112,Z 929.887,A -85,B 0,C 180,E1 18330.103,E2 18330.103} C_VEL
LIN {X 0,Y 446.207,Z 886.049,A -85,B 0,C 180,E1 18338.531,E2 18338.531} C_VEL
LIN {X 0,Y 430.347,Z 856.544,A -85,B 0,C 180,E1 18347.953,E2 18347.953} C_VEL
LIN {X 0,Y 423.283,Z 844.141,A -85,B 0,C 180,E1 18355.571,E2 18355.571} C_VEL
LIN {X 0,Y 421.948,Z 839.151,A -85,B 0,C 180,E1 18360.97,E2 18360.97} C_VEL
LIN {X 0,Y 423.263,Z 843.982,A -85,B 0,C 180,E1 18368.345,E2 18368.345} C_VEL
LIN {X 0,Y 432.034,Z 858.744,A -85,B 0,C 180,E1 18376.912,E2 18376.912} C_VEL
LIN {X 0,Y 447.125,Z 888.671,A -85,B 0,C 180,E1 18385.367,E2 18385.367} C_VEL
LIN {X 0,Y 456.238,Z 919.468,A -85,B 0,C 180,E1 18390.824,E2 18390.824} C_VEL
LIN {X 0,Y 454.936,Z 933.422,A -85,B 0,C 180,E1 18392.106,E2 18392.106} C_VEL
LIN {X 0,Y 431.973,Z 1002.729,A -85,B 0,C 180,E1 18397.191,E2 18397.191} C_VEL
LIN {X 0,Y 406.692,Z 1064.792,A -85,B 0,C 180,E1 18404.573,E2 18404.573} C_VEL
LIN {X 0,Y 384.44,Z 1116.055,A -85,B 0,C 180,E1 18414.263,E2 18414.263} C_VEL
LIN {X 0,Y 369.75,Z 1153.406,A -85,B 0,C 180,E1 18425.704,E2 18425.704} C_VEL
LIN {X 0,Y 364.069,Z 1174.198,A -85,B 0,C 180,E1 18436.683,E2 18436.683} C_VEL
LIN {X 0,Y 363.194,Z 1182.366,A -85,B 0,C 180,E1 18446.343,E2 18446.343} C_VEL
LIN {X 0,Y 363.266,Z 1181.287,A -85,B 0,C 180,E1 18455.93,E2 18455.93} C_VEL
LIN {X 0,Y 365.688,Z 1167.879,A -85,B 0,C 180,E1 18467.392,E2 18467.392} C_VEL
LIN {X 0,Y 374.12,Z 1140.759,A -85,B 0,C 180,E1 18478.788,E2 18478.788} C_VEL
LIN {X 0,Y 392.023,Z 1097.948,A -85,B 0,C 180,E1 18489.614,E2 18489.614} C_VEL
LIN {X 0,Y 415.892,Z 1043.06,A -85,B 0,C 180,E1 18498.327,E2 18498.327} C_VEL
LIN {X 0,Y 419.073,Z 1034.741,A -85,B 0,C 180,E1 18499.393,E2 18499.393} C_VEL
LIN {X 0,Y 384.054,Z 1046.187,A -85,B 0,C 180,E1 18503.741,E2 18503.741} C_VEL
LIN {X 0,Y 371.694,Z 1048.805,A -85,B 0,C 180,E1 18506.291,E2 18506.291} C_VEL
LIN {X 0,Y 368.77,Z 1081.694,A -85,B 0,C 180,E1 18511.169,E2 18511.169} C_VEL
LIN {X 0,Y 367.038,Z 1100.395,A -85,B 0,C 180,E1 18516.952,E2 18516.952} C_VEL
LIN {X 0,Y 367.093,Z 1105.377,A -85,B 0,C 180,E1 18522.015,E2 18522.015} C_VEL
LIN {X 0,Y 368.926,Z 1098.328,A -85,B 0,C 180,E1 18528.204,E2 18528.204} C_VEL
LIN {X 0,Y 371.987,Z 1077.382,A -85,B 0,C 180,E1 18533.629,E2 18533.629} C_VEL
LIN {X 0,Y 374.922,Z 1044.218,A -85,B 0,C 180,E1 18537.749,E2 18537.749} C_VEL
LIN {X 0,Y 376.366,Z 1000.614,A -85,B 0,C 180,E1 18540.14,E2 18540.14} C_VEL
LIN {X 0,Y 377.478,Z 963.845,A -85,B 0,C 180,E1 18541.219,E2 18541.219} C_VEL
LIN {X 0,Y 406.161,Z 898.754,A -85,B 0,C 180,E1 18545.137,E2 18545.137} C_VEL
LIN {X 0,Y 426.654,Z 849.94,A -85,B 0,C 180,E1 18548.843,E2 18548.843} C_VEL
LIN {X 0,Y 438.87,Z 872.511,A -85,B 0,C 180,E1 18557.765,E2 18557.765} C_VEL
LIN {X 0,Y 456.774,Z 910.004,A -85,B 0,C 180,E1 18566.439,E2 18566.439} C_VEL
LIN {X 0,Y 465.264,Z 934.024,A -85,B 0,C 180,E1 18570.304,E2 18570.304} C_VEL
LIN {X 0,Y 443.111,Z 1015.104,A -85,B 0,C 180,E1 18575.011,E2 18575.011} C_VEL
LIN {X 0,Y 420.342,Z 1075.715,A -85,B 0,C 180,E1 18580.885,E2 18580.885} C_VEL
LIN {X 0,Y 397.039,Z 1126.306,A -85,B 0,C 180,E1 18588.836,E2 18588.836} C_VEL
LIN {X 0,Y 377.273,Z 1166.419,A -85,B 0,C 180,E1 18599.222,E2 18599.222} C_VEL
LIN {X 0,Y 366.291,Z 1191.905,A -85,B 0,C 180,E1 18610.713,E2 18610.713} C_VEL
LIN {X 0,Y 363.296,Z 1204.165,A -85,B 0,C 180,E1 18621.659,E2 18621.659} C_VEL
LIN {X 0,Y 363.14,Z 1206.83,A -85,B 0,C 180,E1 18631.261,E2 18631.261} C_VEL
LIN {X 0,Y 363.78,Z 1201.215,A -85,B 0,C 180,E1 18641.98,E2 18641.98} C_VEL
LIN {X 0,Y 369.117,Z 1183.898,A -85,B 0,C 180,E1 18653.696,E2 18653.696} C_VEL
LIN {X 0,Y 383.145,Z 1154.043,A -85,B 0,C 180,E1 18664.622,E2 18664.622} C_VEL
LIN {X 0,Y 404.454,Z 1110.875,A -85,B 0,C 180,E1 18674.03,E2 18674.03} C_VEL
LIN {X 0,Y 428.049,Z 1056.964,A -85,B 0,C 180,E1 18681.249,E2 18681.249} C_VEL
LIN {X 0,Y 432.562,Z 1045.262,A -85,B 0,C 180,E1 18682.427,E2 18682.427} C_VEL
LIN {X 0,Y 436.623,Z 1019.02,A -85,B 0,C 180,E1 18685.534,E2 18685.534} C_VEL
LIN {X 0,Y 458.308,Z 944.11,A -85,B 0,C 180,E1 18690.05,E2 18690.05} C_VEL
LIN {X 0,Y 459.902,Z 934.254,A -85,B 0,C 180,E1 18690.69,E2 18690.69} C_VEL
LIN {X 0,Y 442.547,Z 892.758,A -85,B 0,C 180,E1 18698.839,E2 18698.839} C_VEL
LIN {X 0,Y 427.793,Z 864.166,A -85,B 0,C 180,E1 18708.01,E2 18708.01} C_VEL
LIN {X 0,Y 420.854,Z 851.666,A -85,B 0,C 180,E1 18715.707,E2 18715.707} C_VEL
LIN {X 0,Y 419.735,Z 846.828,A -85,B 0,C 180,E1 18720.975,E2 18720.975} C_VEL
LIN {X 0,Y 421.183,Z 851.996,A -85,B 0,C 180,E1 18728.68,E2 18728.68} C_VEL
LIN {X 0,Y 430.053,Z 867.638,A -85,B 0,C 180,E1 18737.19,E2 18737.19} C_VEL
LIN {X 0,Y 443.771,Z 896.218,A -85,B 0,C 180,E1 18745.238,E2 18745.238} C_VEL
LIN {X 0,Y 451.362,Z 923.989,A -85,B 0,C 180,E1 18750.263,E2 18750.263} C_VEL
LIN {X 0,Y 449.368,Z 938.053,A -85,B 0,C 180,E1 18751.49,E2 18751.49} C_VEL
LIN {X 0,Y 425.83,Z 1006.282,A -85,B 0,C 180,E1 18756.614,E2 18756.614} C_VEL
LIN {X 0,Y 399.673,Z 1067.845,A -85,B 0,C 180,E1 18764.146,E2 18764.146} C_VEL
LIN {X 0,Y 377.096,Z 1117.612,A -85,B 0,C 180,E1 18773.845,E2 18773.845} C_VEL
LIN {X 0,Y 362.268,Z 1153.656,A -85,B 0,C 180,E1 18785.168,E2 18785.168} C_VEL
LIN {X 0,Y 356.16,Z 1174.455,A -85,B 0,C 180,E1 18796.382,E2 18796.382} C_VEL
LIN {X 0,Y 355.195,Z 1182.627,A -85,B 0,C 180,E1 18806.261,E2 18806.261} C_VEL
LIN {X 0,Y 355.287,Z 1181.545,A -85,B 0,C 180,E1 18816.064,E2 18816.064} C_VEL
LIN {X 0,Y 357.804,Z 1168.338,A -85,B 0,C 180,E1 18827.663,E2 18827.663} C_VEL
LIN {X 0,Y 366.742,Z 1141.305,A -85,B 0,C 180,E1 18839.319,E2 18839.319} C_VEL
LIN {X 0,Y 385.125,Z 1099.354,A -85,B 0,C 180,E1 18850.175,E2 18850.175} C_VEL
LIN {X 0,Y 409.732,Z 1045.037,A -85,B 0,C 180,E1 18858.976,E2 18858.976} C_VEL
LIN {X 0,Y 408.113,Z 1043.838,A -85,B 0,C 180,E1 18859.495,E2 18859.495} C_VEL
LIN {X 0,Y 374.478,Z 1053.46,A -85,B 0,C 180,E1 18864.105,E2 18864.105} C_VEL
LIN {X 0,Y 363.365,Z 1055.867,A -85,B 0,C 180,E1 18866.736,E2 18866.736} C_VEL
LIN {X 0,Y 360.666,Z 1086.606,A -85,B 0,C 180,E1 18871.918,E2 18871.918} C_VEL
LIN {X 0,Y 359.052,Z 1103.115,A -85,B 0,C 180,E1 18877.836,E2 18877.836} C_VEL
LIN {X 0,Y 359.635,Z 1105.868,A -85,B 0,C 180,E1 18884.158,E2 18884.158} C_VEL
LIN {X 0,Y 362.229,Z 1093.976,A -85,B 0,C 180,E1 18890.378,E2 18890.378} C_VEL
LIN {X 0,Y 365.457,Z 1068.735,A -85,B 0,C 180,E1 18895.541,E2 18895.541} C_VEL
LIN {X 0,Y 368.497,Z 1030.968,A -85,B 0,C 180,E1 18899.258,E2 18899.258} C_VEL
LIN {X 0,Y 370.331,Z 977.731,A -85,B 0,C 180,E1 18901.483,E2 18901.483} C_VEL
LIN {X 0,Y 397.818,Z 922.235,A -85,B 0,C 180,E1 18905.161,E2 18905.161} C_VEL
LIN {X 0,Y 416.934,Z 876.17,A -85,B 0,C 180,E1 18907.914,E2 18907.914} C_VEL
LIN {X 0,Y 424.813,Z 858.493,A -85,B 0,C 180,E1 18909.395,E2 18909.395} C_VEL
LIN {X 0,Y 437.946,Z 884.184,A -85,B 0,C 180,E1 18918.835,E2 18918.835} C_VEL
LIN {X 0,Y 454.96,Z 922.152,A -85,B 0,C 180,E1 18927.194,E2 18927.194} C_VEL
LIN {X 0,Y 459.588,Z 938.678,A -85,B 0,C 180,E1 18929.681,E2 18929.681} C_VEL
LIN {X 0,Y 437.461,Z 1016.697,A -85,B 0,C 180,E1 18934.307,E2 18934.307} C_VEL
LIN {X 0,Y 414.208,Z 1076.328,A -85,B 0,C 180,E1 18940.174,E2 18940.174} C_VEL
LIN {X 0,Y 389.979,Z 1127.108,A -85,B 0,C 180,E1 18948.297,E2 18948.297} C_VEL
LIN {X 0,Y 370.113,Z 1165.969,A -85,B 0,C 180,E1 18958.559,E2 18958.559} C_VEL
LIN {X 0,Y 358.544,Z 1191.577,A -85,B 0,C 180,E1 18970.28,E2 18970.28} C_VEL
LIN {X 0,Y 355.307,Z 1203.888,A -85,B 0,C 180,E1 18981.47,E2 18981.47} C_VEL
LIN {X 0,Y 355.155,Z 1206.567,A -85,B 0,C 180,E1 18991.289,E2 18991.289} C_VEL
LIN {X 0,Y 355.854,Z 1200.811,A -85,B 0,C 180,E1 19002.376,E2 19002.376} C_VEL
LIN {X 0,Y 361.461,Z 1183.628,A -85,B 0,C 180,E1 19014.179,E2 19014.179} C_VEL
LIN {X 0,Y 376.458,Z 1153.094,A -85,B 0,C 180,E1 19025.483,E2 19025.483} C_VEL
LIN {X 0,Y 399.14,Z 1108.688,A -85,B 0,C 180,E1 19035.136,E2 19035.136} C_VEL
LIN {X 0,Y 423.684,Z 1053.991,A -85,B 0,C 180,E1 19042.364,E2 19042.364} C_VEL
LIN {X 0,Y 436.623,Z 1019.02,A -85,B 0,C 180,E1 19045.534,E2 19045.534} C_VEL
LIN {X 0,Y 440.619,Z 991.219,A -85,B 0,C 180,E1 19048.356,E2 19048.356} C_VEL
LIN {X 0,Y 454.774,Z 938.825,A -85,B 0,C 180,E1 19051.25,E2 19051.25} C_VEL
LIN {X 0,Y 437.953,Z 897.383,A -85,B 0,C 180,E1 19059.668,E2 19059.668} C_VEL
LIN {X 0,Y 423.616,Z 868.87,A -85,B 0,C 180,E1 19069.405,E2 19069.405} C_VEL
LIN {X 0,Y 417.666,Z 854.712,A -85,B 0,C 180,E1 19079.679,E2 19079.679} C_VEL
LIN {X 0,Y 418.058,Z 857.83,A -85,B 0,C 180,E1 19086.864,E2 19086.864} C_VEL
LIN {X 0,Y 424.456,Z 869.865,A -85,B 0,C 180,E1 19094.825,E2 19094.825} C_VEL
LIN {X 0,Y 436.636,Z 894.293,A -85,B 0,C 180,E1 19102.895,E2 19102.895} C_VEL
LIN {X 0,Y 446.447,Z 926.685,A -85,B 0,C 180,E1 19109.458,E2 19109.458} C_VEL
LIN {X 0,Y 444.515,Z 940.564,A -85,B 0,C 180,E1 19110.734,E2 19110.734} C_VEL
LIN {X 0,Y 420.249,Z 1008.458,A -85,B 0,C 180,E1 19115.897,E2 19115.897} C_VEL
LIN {X 0,Y 393.125,Z 1069.917,A -85,B 0,C 180,E1 19123.555,E2 19123.555} C_VEL
LIN {X 0,Y 369.78,Z 1119.17,A -85,B 0,C 180,E1 19133.411,E2 19133.411} C_VEL
LIN {X 0,Y 354.173,Z 1155.446,A -85,B 0,C 180,E1 19145.238,E2 19145.238} C_VEL
LIN {X 0,Y 348.289,Z 1174.714,A -85,B 0,C 180,E1 19156.068,E2 19156.068} C_VEL
LIN {X 0,Y 347.191,Z 1182.889,A -85,B 0,C 180,E1 19166.175,E2 19166.175} C_VEL
LIN {X 0,Y 347.293,Z 1181.805,A -85,B 0,C 180,E1 19176.204,E2 19176.204} C_VEL
LIN {X 0,Y 349.972,Z 1168.604,A -85,B 0,C 180,E1 19188.071,E2 19188.071} C_VEL
LIN {X 0,Y 359.201,Z 1142.326,A -85,B 0,C 180,E1 19199.721,E2 19199.721} C_VEL
LIN {X 0,Y 378.267,Z 1100.765,A -85,B 0,C 180,E1 19210.757,E2 19210.757} C_VEL
LIN {X 0,Y 400.545,Z 1051.276,A -85,B 0,C 180,E1 19219.284,E2 19219.284} C_VEL
LIN {X 0,Y 360.645,Z 1060.583,A -85,B 0,C 180,E1 19225.478,E2 19225.478} C_VEL
LIN {X 0,Y 354.982,Z 1061.88,A -85,B 0,C 180,E1 19227.169,E2 19227.169} C_VEL
LIN {X 0,Y 352.52,Z 1090.099,A -85,B 0,C 180,E1 19232.453,E2 19232.453} C_VEL
LIN {X 0,Y 351.065,Z 1105.132,A -85,B 0,C 180,E1 19238.525,E2 19238.525} C_VEL
LIN {X 0,Y 351.647,Z 1107.345,A -85,B 0,C 180,E1 19243.788,E2 19243.788} C_VEL
LIN {X 0,Y 354.296,Z 1096.615,A -85,B 0,C 180,E1 19250.23,E2 19250.23} C_VEL
LIN {X 0,Y 357.728,Z 1072.151,A -85,B 0,C 180,E1 19255.627,E2 19255.627} C_VEL
LIN {X 0,Y 361.09,Z 1035.104,A -85,B 0,C 180,E1 19259.544,E2 19259.544} C_VEL
LIN {X 0,Y 363.163,Z 990.541,A -85,B 0,C 180,E1 19261.758,E2 19261.758} C_VEL
LIN {X 0,Y 394.066,Z 933.682,A -85,B 0,C 180,E1 19265.854,E2 19265.854} C_VEL
LIN {X 0,Y 416.129,Z 881.912,A -85,B 0,C 180,E1 19268.702,E2 19268.702} C_VEL
LIN {X 0,Y 423.07,Z 867.237,A -85,B 0,C 180,E1 19270.032,E2 19270.032} C_VEL
LIN {X 0,Y 436.831,Z 895.836,A -85,B 0,C 180,E1 19279.857,E2 19279.857} C_VEL
LIN {X 0,Y 453.83,Z 937.006,A -85,B 0,C 180,E1 19288.401,E2 19288.401} C_VEL
LIN {X 0,Y 452.912,Z 946.848,A -85,B 0,C 180,E1 19289.208,E2 19289.208} C_VEL
LIN {X 0,Y 430.549,Z 1022.13,A -85,B 0,C 180,E1 19293.88,E2 19293.88} C_VEL
LIN {X 0,Y 405.939,Z 1081.802,A -85,B 0,C 180,E1 19300.069,E2 19300.069} C_VEL
LIN {X 0,Y 380.799,Z 1132.01,A -85,B 0,C 180,E1 19308.633,E2 19308.633} C_VEL
LIN {X 0,Y 360.736,Z 1169.493,A -85,B 0,C 180,E1 19319.301,E2 19319.301} C_VEL
LIN {X 0,Y 350.001,Z 1193.195,A -85,B 0,C 180,E1 19331.096,E2 19331.096} C_VEL
LIN {X 0,Y 347.307,Z 1203.612,A -85,B 0,C 180,E1 19341.272,E2 19341.272} C_VEL
LIN {X 0,Y 347.153,Z 1206.304,A -85,B 0,C 180,E1 19351.319,E2 19351.319} C_VEL
LIN {X 0,Y 347.911,Z 1200.524,A -85,B 0,C 180,E1 19362.663,E2 19362.663} C_VEL
LIN {X 0,Y 353.853,Z 1183.337,A -85,B 0,C 180,E1 19374.691,E2 19374.691} C_VEL
LIN {X 0,Y 369.636,Z 1152.581,A -85,B 0,C 180,E1 19386.24,E2 19386.24} C_VEL
LIN {X 0,Y 393.062,Z 1108.324,A -85,B 0,C 180,E1 19395.96,E2 19395.96} C_VEL
LIN {X 0,Y 418.361,Z 1053.602,A -85,B 0,C 180,E1 19403.241,E2 19403.241} C_VEL
LIN {X 0,Y 440.619,Z 991.219,A -85,B 0,C 180,E1 19408.356,E2 19408.356} C_VEL
LIN {X 0,Y 444.713,Z 961.842,A -85,B 0,C 180,E1 19410.887,E2 19410.887} C_VEL
LIN {X 0,Y 449.345,Z 942.498,A -85,B 0,C 180,E1 19411.979,E2 19411.979} C_VEL
LIN {X 0,Y 433.349,Z 902.091,A -85,B 0,C 180,E1 19420.51,E2 19420.51} C_VEL
LIN {X 0,Y 419.996,Z 873.955,A -85,B 0,C 180,E1 19430.583,E2 19430.583} C_VEL
LIN {X 0,Y 415.156,Z 862.129,A -85,B 0,C 180,E1 19440.986,E2 19440.986} C_VEL
LIN {X 0,Y 417.808,Z 868.538,A -85,B 0,C 180,E1 19450.135,E2 19450.135} C_VEL
LIN {X 0,Y 428.68,Z 890.343,A -85,B 0,C 180,E1 19459.585,E2 19459.585} C_VEL
LIN {X 0,Y 439.827,Z 921.861,A -85,B 0,C 180,E1 19467.197,E2 19467.197} C_VEL
LIN {X 0,Y 441.038,Z 938.837,A -85,B 0,C 180,E1 19469.701,E2 19469.701} C_VEL
LIN {X 0,Y 415.637,Z 1008.447,A -85,B 0,C 180,E1 19474.951,E2 19474.951} C_VEL
LIN {X 0,Y 387.444,Z 1070.247,A -85,B 0,C 180,E1 19482.664,E2 19482.664} C_VEL
LIN {X 0,Y 363.157,Z 1119.473,A -85,B 0,C 180,E1 19492.631,E2 19492.631} C_VEL
LIN {X 0,Y 346.66,Z 1155.866,A -85,B 0,C 180,E1 19504.736,E2 19504.736} C_VEL
LIN {X 0,Y 340.396,Z 1174.977,A -85,B 0,C 180,E1 19515.738,E2 19515.738} C_VEL
LIN {X 0,Y 339.197,Z 1183.151,A -85,B 0,C 180,E1 19526.084,E2 19526.084} C_VEL
LIN {X 0,Y 339.299,Z 1182.066,A -85,B 0,C 180,E1 19536.351,E2 19536.351} C_VEL
LIN {X 0,Y 342.112,Z 1169.041,A -85,B 0,C 180,E1 19548.392,E2 19548.392} C_VEL
LIN {X 0,Y 352.46,Z 1141.59,A -85,B 0,C 180,E1 19560.725,E2 19560.725} C_VEL
LIN {X 0,Y 373.132,Z 1098.896,A -85,B 0,C 180,E1 19572.059,E2 19572.059} C_VEL
LIN {X 0,Y 392.071,Z 1058.56,A -85,B 0,C 180,E1 19579.186,E2 19579.186} C_VEL
LIN {X 0,Y 356.001,Z 1066.221,A -85,B 0,C 180,E1 19584.963,E2 19584.963} C_VEL
LIN {X 0,Y 346.487,Z 1068,A -85,B 0,C 180,E1 19587.697,E2 19587.697} C_VEL
LIN {X 0,Y 344.279,Z 1093.881,A -85,B 0,C 180,E1 19593.11,E2 19593.11} C_VEL
LIN {X 0,Y 343.121,Z 1107.201,A -85,B 0,C 180,E1 19599.362,E2 19599.362} C_VEL
LIN {X 0,Y 344.399,Z 1106.786,A -85,B 0,C 180,E1 19606.054,E2 19606.054} C_VEL
LIN {X 0,Y 347.663,Z 1092.08,A -85,B 0,C 180,E1 19612.236,E2 19612.236} C_VEL
LIN {X 0,Y 351.43,Z 1063.353,A -85,B 0,C 180,E1 19617.443,E2 19617.443} C_VEL
LIN {X 0,Y 354.287,Z 1023.669,A -85,B 0,C 180,E1 19620.839,E2 19620.839} C_VEL
LIN {X 0,Y 355.816,Z 1002.612,A -85,B 0,C 180,E1 19621.98,E2 19621.98} C_VEL
LIN {X 0,Y 388.325,Z 948.347,A -85,B 0,C 180,E1 19626.256,E2 19626.256} C_VEL
LIN {X 0,Y 416.094,Z 886.099,A -85,B 0,C 180,E1 19629.639,E2 19629.639} C_VEL
LIN {X 0,Y 420.81,Z 876.129,A -85,B 0,C 180,E1 19630.448,E2 19630.448} C_VEL
LIN {X 0,Y 433.739,Z 903.715,A -85,B 0,C 180,E1 19639.848,E2 19639.848} C_VEL
LIN {X 0,Y 449.416,Z 943.608,A -85,B 0,C 180,E1 19648.173,E2 19648.173} C_VEL
LIN {X 0,Y 427.037,Z 1018.121,A -85,B 0,C 180,E1 19652.695,E2 19652.695} C_VEL
LIN {X 0,Y 401.336,Z 1079.312,A -85,B 0,C 180,E1 19658.909,E2 19658.909} C_VEL
LIN {X 0,Y 375.604,Z 1129.298,A -85,B 0,C 180,E1 19667.303,E2 19667.303} C_VEL
LIN {X 0,Y 354.331,Z 1167.81,A -85,B 0,C 180,E1 19678.152,E2 19678.152} C_VEL
LIN {X 0,Y 342.224,Z 1192.864,A -85,B 0,C 180,E1 19690.649,E2 19690.649} C_VEL
LIN {X 0,Y 339.333,Z 1203.334,A -85,B 0,C 180,E1 19701.065,E2 19701.065} C_VEL
LIN {X 0,Y 339.166,Z 1206.041,A -85,B 0,C 180,E1 19711.35,E2 19711.35} C_VEL
LIN {X 0,Y 339.963,Z 1200.234,A -85,B 0,C 180,E1 19722.964,E2 19722.964} C_VEL
LIN {X 0,Y 346.519,Z 1182.542,A -85,B 0,C 180,E1 19735.481,E2 19735.481} C_VEL
LIN {X 0,Y 363.449,Z 1151.03,A -85,B 0,C 180,E1 19747.334,E2 19747.334} C_VEL
LIN {X 0,Y 388.282,Z 1105.625,A -85,B 0,C 180,E1 19757.202,E2 19757.202} C_VEL
LIN {X 0,Y 414.427,Z 1050.238,A -85,B 0,C 180,E1 19764.44,E2 19764.44} C_VEL
LIN {X 0,Y 437.303,Z 986.957,A -85,B 0,C 180,E1 19769.496,E2 19769.496} C_VEL
LIN {X 0,Y 444.713,Z 961.842,A -85,B 0,C 180,E1 19770.887,E2 19770.887} C_VEL
LIN {X 0,Y 444.94,Z 948.195,A -85,B 0,C 180,E1 19772.307,E2 19772.307} C_VEL
LIN {X 0,Y 441.127,Z 937.857,A -85,B 0,C 180,E1 19774.281,E2 19774.281} C_VEL
LIN {X 0,Y 427.305,Z 903.463,A -85,B 0,C 180,E1 19782.371,E2 19782.371} C_VEL
LIN {X 0,Y 416.497,Z 880.208,A -85,B 0,C 180,E1 19791.559,E2 19791.559} C_VEL
LIN {X 0,Y 412.767,Z 869.764,A -85,B 0,C 180,E1 19800.991,E2 19800.991} C_VEL
LIN {X 0,Y 414.914,Z 875.647,A -85,B 0,C 180,E1 19809.409,E2 19809.409} C_VEL
LIN {X 0,Y 424.204,Z 894.728,A -85,B 0,C 180,E1 19818.409,E2 19818.409} C_VEL
LIN {X 0,Y 434.541,Z 924.366,A -85,B 0,C 180,E1 19826.091,E2 19826.091} C_VEL
LIN {X 0,Y 436.7,Z 940.376,A -85,B 0,C 180,E1 19828.852,E2 19828.852} C_VEL
LIN {X 0,Y 410.661,Z 1009.57,A -85,B 0,C 180,E1 19834.091,E2 19834.091} C_VEL
LIN {X 0,Y 381.794,Z 1070.757,A -85,B 0,C 180,E1 19841.783,E2 19841.783} C_VEL
LIN {X 0,Y 356.624,Z 1119.781,A -85,B 0,C 180,E1 19851.825,E2 19851.825} C_VEL
LIN {X 0,Y 339.177,Z 1156.257,A -85,B 0,C 180,E1 19864.195,E2 19864.195} C_VEL
LIN {X 0,Y 332.518,Z 1175.243,A -85,B 0,C 180,E1 19875.393,E2 19875.393} C_VEL
LIN {X 0,Y 331.192,Z 1183.413,A -85,B 0,C 180,E1 19885.99,E2 19885.99} C_VEL
LIN {X 0,Y 331.306,Z 1182.327,A -85,B 0,C 180,E1 19896.504,E2 19896.504} C_VEL
LIN {X 0,Y 334.353,Z 1169.14,A -85,B 0,C 180,E1 19908.946,E2 19908.946} C_VEL
LIN {X 0,Y 345.248,Z 1142.016,A -85,B 0,C 180,E1 19921.384,E2 19921.384} C_VEL
LIN {X 0,Y 367.018,Z 1099.238,A -85,B 0,C 180,E1 19932.926,E2 19932.926} C_VEL
LIN {X 0,Y 384.085,Z 1065.399,A -85,B 0,C 180,E1 19939.04,E2 19939.04} C_VEL
LIN {X 0,Y 351.296,Z 1071.768,A -85,B 0,C 180,E1 19944.423,E2 19944.423} C_VEL
LIN {X 0,Y 338.335,Z 1073.396,A -85,B 0,C 180,E1 19948.209,E2 19948.209} C_VEL
LIN {X 0,Y 335.981,Z 1097.954,A -85,B 0,C 180,E1 19954.03,E2 19954.03} C_VEL
LIN {X 0,Y 335.244,Z 1109.065,A -85,B 0,C 180,E1 19960.238,E2 19960.238} C_VEL
LIN {X 0,Y 336.862,Z 1107.051,A -85,B 0,C 180,E1 19967.063,E2 19967.063} C_VEL
LIN {X 0,Y 340.573,Z 1090.378,A -85,B 0,C 180,E1 19973.36,E2 19973.36} C_VEL
LIN {X 0,Y 344.605,Z 1059.803,A -85,B 0,C 180,E1 19978.497,E2 19978.497} C_VEL
LIN {X 0,Y 347.441,Z 1018.25,A -85,B 0,C 180,E1 19981.743,E2 19981.743} C_VEL
LIN {X 0,Y 383.645,Z 959.954,A -85,B 0,C 180,E1 19986.874,E2 19986.874} C_VEL
LIN {X 0,Y 416.762,Z 889.117,A -85,B 0,C 180,E1 19990.683,E2 19990.683} C_VEL
LIN {X 0,Y 418.729,Z 885.221,A -85,B 0,C 180,E1 19991.028,E2 19991.028} C_VEL
LIN {X 0,Y 431.414,Z 913.505,A -85,B 0,C 180,E1 20000.339,E2 20000.339} C_VEL
LIN {X 0,Y 443.797,Z 948.895,A -85,B 0,C 180,E1 20007.551,E2 20007.551} C_VEL
LIN {X 0,Y 421.143,Z 1020.889,A -85,B 0,C 180,E1 20012.033,E2 20012.033} C_VEL
LIN {X 0,Y 395.207,Z 1080.238,A -85,B 0,C 180,E1 20018.182,E2 20018.182} C_VEL
LIN {X 0,Y 368.408,Z 1130.434,A -85,B 0,C 180,E1 20026.793,E2 20026.793} C_VEL
LIN {X 0,Y 346.873,Z 1168.029,A -85,B 0,C 180,E1 20037.668,E2 20037.668} C_VEL
LIN {X 0,Y 334.473,Z 1192.528,A -85,B 0,C 180,E1 20050.182,E2 20050.182} C_VEL
LIN {X 0,Y 331.339,Z 1203.054,A -85,B 0,C 180,E1 20060.847,E2 20060.847} C_VEL
LIN {X 0,Y 331.162,Z 1205.777,A -85,B 0,C 180,E1 20071.382,E2 20071.382} C_VEL
LIN {X 0,Y 332.039,Z 1199.943,A -85,B 0,C 180,E1 20083.279,E2 20083.279} C_VEL
LIN {X 0,Y 339.039,Z 1182.163,A -85,B 0,C 180,E1 20096.085,E2 20096.085} C_VEL
LIN {X 0,Y 356.792,Z 1150.503,A -85,B 0,C 180,E1 20108.154,E2 20108.154} C_VEL
LIN {X 0,Y 382.516,Z 1105.059,A -85,B 0,C 180,E1 20118.113,E2 20118.113} C_VEL
LIN {X 0,Y 409.52,Z 1049.496,A -85,B 0,C 180,E1 20125.392,E2 20125.392} C_VEL
LIN {X 0,Y 432.719,Z 987.34,A -85,B 0,C 180,E1 20130.362,E2 20130.362} C_VEL
LIN {X 0,Y 444.016,Z 946.1,A -85,B 0,C 180,E1 20132.739,E2 20132.739} C_VEL
LIN {X 0,Y 441.127,Z 937.857,A -85,B 0,C 180,E1 20134.281,E2 20134.281} C_VEL
LIN {X 0,Y 430.284,Z 926.049,A -85,B 0,C 180,E1 20138.468,E2 20138.468} C_VEL
LIN {X 0,Y 417.629,Z 896.296,A -85,B 0,C 180,E1 20147.564,E2 20147.564} C_VEL
LIN {X 0,Y 411.841,Z 883.159,A -85,B 0,C 180,E1 20154.653,E2 20154.653} C_VEL
LIN {X 0,Y 410.406,Z 877.46,A -85,B 0,C 180,E1 20163.117,E2 20163.117} C_VEL
LIN {X 0,Y 415.424,Z 889.164,A -85,B 0,C 180,E1 20172.998,E2 20172.998} C_VEL
LIN {X 0,Y 425.722,Z 914.287,A -85,B 0,C 180,E1 20181.911,E2 20181.911} C_VEL
LIN {X 0,Y 432.112,Z 942.857,A -85,B 0,C 180,E1 20188.038,E2 20188.038} C_VEL
LIN {X 0,Y 405.473,Z 1011.476,A -85,B 0,C 180,E1 20193.284,E2 20193.284} C_VEL
LIN {X 0,Y 375.37,Z 1072.968,A -85,B 0,C 180,E1 20201.139,E2 20201.139} C_VEL
LIN {X 0,Y 349.427,Z 1121.333,A -85,B 0,C 180,E1 20211.317,E2 20211.317} C_VEL
LIN {X 0,Y 331.212,Z 1157.767,A -85,B 0,C 180,E1 20224.124,E2 20224.124} C_VEL
LIN {X 0,Y 324.27,Z 1177.081,A -85,B 0,C 180,E1 20236.396,E2 20236.396} C_VEL
LIN {X 0,Y 323.201,Z 1183.675,A -85,B 0,C 180,E1 20245.89,E2 20245.89} C_VEL
LIN {X 0,Y 323.324,Z 1182.589,A -85,B 0,C 180,E1 20256.666,E2 20256.666} C_VEL
LIN {X 0,Y 326.388,Z 1170.139,A -85,B 0,C 180,E1 20268.915,E2 20268.915} C_VEL
LIN {X 0,Y 337.731,Z 1143.269,A -85,B 0,C 180,E1 20281.78,E2 20281.78} C_VEL
LIN {X 0,Y 360.298,Z 1100.796,A -85,B 0,C 180,E1 20293.559,E2 20293.559} C_VEL
LIN {X 0,Y 374.542,Z 1072.235,A -85,B 0,C 180,E1 20299.099,E2 20299.099} C_VEL
LIN {X 0,Y 336.177,Z 1077.712,A -85,B 0,C 180,E1 20306.491,E2 20306.491} C_VEL
LIN {X 0,Y 330.001,Z 1079.334,A -85,B 0,C 180,E1 20308.943,E2 20308.943} C_VEL
LIN {X 0,Y 327.775,Z 1101.556,A -85,B 0,C 180,E1 20314.933,E2 20314.933} C_VEL
LIN {X 0,Y 327.504,Z 1110.917,A -85,B 0,C 180,E1 20321.539,E2 20321.539} C_VEL
LIN {X 0,Y 329.441,Z 1106.995,A -85,B 0,C 180,E1 20328.118,E2 20328.118} C_VEL
LIN {X 0,Y 333.549,Z 1088.684,A -85,B 0,C 180,E1 20334.465,E2 20334.465} C_VEL
LIN {X 0,Y 337.741,Z 1057.49,A -85,B 0,C 180,E1 20339.432,E2 20339.432} C_VEL
LIN {X 0,Y 341.29,Z 1024.006,A -85,B 0,C 180,E1 20342.371,E2 20342.371} C_VEL
LIN {X 0,Y 372.346,Z 981.427,A -85,B 0,C 180,E1 20346.702,E2 20346.702} C_VEL
LIN {X 0,Y 405.997,Z 916.986,A -85,B 0,C 180,E1 20350.278,E2 20350.278} C_VEL
LIN {X 0,Y 416.64,Z 894.225,A -85,B 0,C 180,E1 20351.616,E2 20351.616} C_VEL
LIN {X 0,Y 429.228,Z 924.21,A -85,B 0,C 180,E1 20361.034,E2 20361.034} C_VEL
LIN {X 0,Y 438.383,Z 953.388,A -85,B 0,C 180,E1 20366.852,E2 20366.852} C_VEL
LIN {X 0,Y 415.274,Z 1023.751,A -85,B 0,C 180,E1 20371.356,E2 20371.356} C_VEL
LIN {X 0,Y 388.013,Z 1083.45,A -85,B 0,C 180,E1 20377.736,E2 20377.736} C_VEL
LIN {X 0,Y 359.917,Z 1133.834,A -85,B 0,C 180,E1 20386.788,E2 20386.788} C_VEL
LIN {X 0,Y 337.729,Z 1170.86,A -85,B 0,C 180,E1 20398.217,E2 20398.217} C_VEL
LIN {X 0,Y 325.964,Z 1193.949,A -85,B 0,C 180,E1 20411.058,E2 20411.058} C_VEL
LIN {X 0,Y 323.135,Z 1204.161,A -85,B 0,C 180,E1 20423.33,E2 20423.33} C_VEL
LIN {X 0,Y 323.159,Z 1205.513,A -85,B 0,C 180,E1 20431.417,E2 20431.417} C_VEL
LIN {X 0,Y 324.089,Z 1199.649,A -85,B 0,C 180,E1 20443.611,E2 20443.611} C_VEL
LIN {X 0,Y 331.476,Z 1181.947,A -85,B 0,C 180,E1 20456.632,E2 20456.632} C_VEL
LIN {X 0,Y 350.213,Z 1149.96,A -85,B 0,C 180,E1 20469.004,E2 20469.004} C_VEL
LIN {X 0,Y 376.773,Z 1104.661,A -85,B 0,C 180,E1 20479.032,E2 20479.032} C_VEL
LIN {X 0,Y 405.043,Z 1048.082,A -85,B 0,C 180,E1 20486.443,E2 20486.443} C_VEL
LIN {X 0,Y 429.237,Z 984.693,A -85,B 0,C 180,E1 20491.43,E2 20491.43} C_VEL
LIN {X 0,Y 439.126,Z 951.216,A -85,B 0,C 180,E1 20493.24,E2 20493.24} C_VEL
LIN {X 0,Y 430.284,Z 926.049,A -85,B 0,C 180,E1 20498.468,E2 20498.468} C_VEL
LIN {X 0,Y 420.35,Z 917.292,A -85,B 0,C 180,E1 20502.934,E2 20502.934} C_VEL
LIN {X 0,Y 410.537,Z 894.063,A -85,B 0,C 180,E1 20512.505,E2 20512.505} C_VEL
LIN {X 0,Y 407.987,Z 885.122,A -85,B 0,C 180,E1 20523.135,E2 20523.135} C_VEL
LIN {X 0,Y 412.944,Z 897.486,A -85,B 0,C 180,E1 20533.177,E2 20533.177} C_VEL
LIN {X 0,Y 421.918,Z 920.855,A -85,B 0,C 180,E1 20541.574,E2 20541.574} C_VEL
LIN {X 0,Y 427.073,Z 946.97,A -85,B 0,C 180,E1 20547.314,E2 20547.314} C_VEL
LIN {X 0,Y 399.882,Z 1014.384,A -85,B 0,C 180,E1 20552.554,E2 20552.554} C_VEL
LIN {X 0,Y 369.198,Z 1074.783,A -85,B 0,C 180,E1 20560.412,E2 20560.412} C_VEL
LIN {X 0,Y 342.369,Z 1122.699,A -85,B 0,C 180,E1 20570.736,E2 20570.736} C_VEL
LIN {X 0,Y 323.823,Z 1158.043,A -85,B 0,C 180,E1 20583.488,E2 20583.488} C_VEL
LIN {X 0,Y 316.377,Z 1177.346,A -85,B 0,C 180,E1 20596.05,E2 20596.05} C_VEL
LIN {X 0,Y 315.196,Z 1183.938,A -85,B 0,C 180,E1 20605.786,E2 20605.786} C_VEL
LIN {X 0,Y 315.332,Z 1182.852,A -85,B 0,C 180,E1 20616.836,E2 20616.836} C_VEL
LIN {X 0,Y 318.611,Z 1170.421,A -85,B 0,C 180,E1 20629.396,E2 20629.396} C_VEL
LIN {X 0,Y 330.7,Z 1143.564,A -85,B 0,C 180,E1 20642.541,E2 20642.541} C_VEL
LIN {X 0,Y 354.219,Z 1101.323,A -85,B 0,C 180,E1 20654.451,E2 20654.451} C_VEL
LIN {X 0,Y 366.585,Z 1079.528,A -85,B 0,C 180,E1 20658.663,E2 20658.663} C_VEL
LIN {X 0,Y 325.587,Z 1082.986,A -85,B 0,C 180,E1 20667.687,E2 20667.687} C_VEL
LIN {X 0,Y 321.711,Z 1084.513,A -85,B 0,C 180,E1 20669.628,E2 20669.628} C_VEL
LIN {X 0,Y 319.572,Z 1105.733,A -85,B 0,C 180,E1 20676.286,E2 20676.286} C_VEL
LIN {X 0,Y 319.682,Z 1112.247,A -85,B 0,C 180,E1 20682.115,E2 20682.115} C_VEL
LIN {X 0,Y 322.18,Z 1106.846,A -85,B 0,C 180,E1 20689.223,E2 20689.223} C_VEL
LIN {X 0,Y 326.498,Z 1087.159,A -85,B 0,C 180,E1 20695.541,E2 20695.541} C_VEL
LIN {X 0,Y 330.963,Z 1054.957,A -85,B 0,C 180,E1 20700.405,E2 20700.405} C_VEL
LIN {X 0,Y 333.769,Z 1033.999,A -85,B 0,C 180,E1 20702.424,E2 20702.424} C_VEL
LIN {X 0,Y 362.399,Z 998.527,A -85,B 0,C 180,E1 20706.802,E2 20706.802} C_VEL
LIN {X 0,Y 397.358,Z 939.732,A -85,B 0,C 180,E1 20710.43,E2 20710.43} C_VEL
LIN {X 0,Y 413.931,Z 904.28,A -85,B 0,C 180,E1 20712.143,E2 20712.143} C_VEL
LIN {X 0,Y 424.186,Z 927.619,A -85,B 0,C 180,E1 20719.929,E2 20719.929} C_VEL
LIN {X 0,Y 433.208,Z 957.133,A -85,B 0,C 180,E1 20726.108,E2 20726.108} C_VEL
LIN {X 0,Y 409.332,Z 1026.797,A -85,B 0,C 180,E1 20730.678,E2 20730.678} C_VEL
LIN {X 0,Y 381.594,Z 1085.107,A -85,B 0,C 180,E1 20737.066,E2 20737.066} C_VEL
LIN {X 0,Y 352.874,Z 1134.691,A -85,B 0,C 180,E1 20746.194,E2 20746.194} C_VEL
LIN {X 0,Y 329.635,Z 1172.016,A -85,B 0,C 180,E1 20758.121,E2 20758.121} C_VEL
LIN {X 0,Y 318.21,Z 1193.626,A -85,B 0,C 180,E1 20770.578,E2 20770.578} C_VEL
